# B&R Automation Studio project Nitto (part 8)

#### gunwfeedi.ax
```
InitParameter (Version=2.37.0, NcSwId=ACP10)
  ACP10AXIS_typ:
    dig_in:
      level:
        reference = ncACTIV_HI
        pos_hw_end = ncACTIV_HI
        neg_hw_end = ncACTIV_HI
        trigger1 = ncACTIV_HI
        trigger2 = ncACTIV_HI
    encoder_if:
      parameter:
        count_dir = ncSTANDARD
        scaling:
          load:
            units = 118000
            rev_motor = 83
    limit:
      parameter:
        v_pos = 75000.0
        v_neg = 75000.0
        a1_pos = 550000.0
        a2_pos = 550000.0
        a1_neg = 550000.0
        a2_neg = 550000.0
        t_jolt = 0.0
        t_in_pos = 0.0
        pos_sw_end = 2000000000
        neg_sw_end = -2000000000
        ds_warning = 1500.0
        ds_stop = 3000.0
        a_stop = 1.0e+30
        dv_stop = 0.0
        dv_stop_mode = ncOFF
    controller:
      mode = ncPOSITION
      position:
        kv = 50.0
        tn = 0.0
        t_predict = 0.002
        t_total = 0.002
        p_max = 1.0e+30
        i_max = 0.0
      speed:
        kv = 2.0
        tn = 0.0
        t_filter = 0.0
        isq_filter1:
          type = ncOFF
          a0 = 0.0
          a1 = 0.0
          b0 = 0.0
          b1 = 0.0
          b2 = 0.0
          c0_par_id = 0
          c1_par_id = 0
        isq_filter2:
          type = ncOFF
          a0 = 0.0
          a1 = 0.0
          b0 = 0.0
          b1 = 0.0
          b2 = 0.0
          c0_par_id = 0
          c1_par_id = 0
        isq_filter3:
          type = ncOFF
          a0 = 0.0
          a1 = 0.0
          b0 = 0.0
          b1 = 0.0
          b2 = 0.0
          c0_par_id = 0
          c1_par_id = 0
      uf:
        type = ncLINEAR
        auto_config = ncMOTOR_PAR
        u0 = 0.0
        un = 0.0
        fn = 50.0
        k_f_slip = 0.0
      ff:
        torque_load = 0.0
        torque_pos = 0.0
        torque_neg = 0.0
        kv_torque = 0.0
        inertia = 0.0
        t_filter_a = 0.0
    move:
      stop:
        parameter[0]:
          decel_ramp = ncA_LIMIT
          controller = ncON
        parameter[1]:
          decel_ramp = ncA_LIMIT
          controller = ncON
        parameter[2]:
          decel_ramp = ncA_LIMIT
          controller = ncON
        parameter[3]:
          decel_ramp = ncA_LIMIT
          controller = ncON
        quickstop:
          decel_ramp = ncA_LIMIT
        drive_error:
          decel_ramp = ncA_LIMIT
      homing:
        parameter:
          s = 0
          v_switch = 5000.0
          v_trigger = 500.0
          a = 50000.0
          mode = ncDIRECT
          edge_sw = ncPOSITIVE
          start_dir = ncPOSITIVE
          trigg_dir = ncPOSITIVE
          ref_pulse = ncOFF
          fix_dir = ncOFF
          tr_s_block = 0.0
          torque_lim = 0.0
          ds_block = 0.0
          ds_stop = 0.0
      basis:
        parameter:
          v_pos = 5000.0
          v_neg = 5000.0
          a1_pos = 100000.0
          a2_pos = 100000.0
          a1_neg = 100000.0
          a2_neg = 100000.0
    message:
      text:
        parameter:
          format = ncBREAK
          columns = 80
          data_modul = acp10etxen
```

### Data object Logical/AxisObj/ggrid1i (Ax)

#### ggrid1i.ax
```
InitParameter (Version=2.37.0, NcSwId=ACP10)
  ACP10AXIS_typ:
    dig_in:
      level:
        reference = ncACTIV_HI
        pos_hw_end = ncACTIV_HI
        neg_hw_end = ncACTIV_HI
        trigger1 = ncACTIV_HI
        trigger2 = ncACTIV_HI
    encoder_if:
      parameter:
        count_dir = ncSTANDARD
        scaling:
          load:
            units = 792000
            rev_motor = 2880
    limit:
      parameter:
        v_pos = 13750.0
        v_neg = 13750.0
        a1_pos = 46000.0
        a2_pos = 46000.0
        a1_neg = 46000.0
        a2_neg = 46000.0
        t_jolt = 0.0
        t_in_pos = 0.0
        pos_sw_end = 2000000000
        neg_sw_end = -2000000000
        ds_warning = 500.0
        ds_stop = 1000.0
        a_stop = 1.0e+30
        dv_stop = 0.0
        dv_stop_mode = ncOFF
    controller:
      mode = ncPOSITION
      position:
        kv = 180.0
        tn = 0.0
        t_predict = 0.0004
        t_total = 0.0004
        p_max = 1.0e+30
        i_max = 0.0
      speed:
        kv = 3.35
        tn = 0.0
        t_filter = 0.0
        isq_filter1:
          type = ncOFF
          a0 = 0.0
          a1 = 0.0
          b0 = 0.0
          b1 = 0.0
          b2 = 0.0
          c0_par_id = 0
          c1_par_id = 0
        isq_filter2:
          type = ncOFF
          a0 = 0.0
          a1 = 0.0
          b0 = 0.0
          b1 = 0.0
          b2 = 0.0
          c0_par_id = 0
          c1_par_id = 0
        isq_filter3:
          type = ncOFF
          a0 = 0.0
          a1 = 0.0
          b0 = 0.0
          b1 = 0.0
          b2 = 0.0
          c0_par_id = 0
          c1_par_id = 0
      uf:
        type = ncLINEAR
        auto_config = ncMOTOR_PAR
        u0 = 0.0
        un = 0.0
        fn = 50.0
        k_f_slip = 0.0
      ff:
        torque_load = 0.0
        torque_pos = 0.0
        torque_neg = 0.0
        kv_torque = 0.0
        inertia = 0.0
        t_filter_a = 0.0
    move:
      stop:
        parameter[0]:
          decel_ramp = ncA_LIMIT
          controller = ncON
        parameter[1]:
          decel_ramp = ncA_LIMIT
          controller = ncON
        parameter[2]:
          decel_ramp = ncA_LIMIT
          controller = ncON
        parameter[3]:
          decel_ramp = ncA_LIMIT
          controller = ncON
        quickstop:
          decel_ramp = ncA_LIMIT
        drive_error:
          decel_ramp = ncA_LIMIT
      homing:
        parameter:
          s = 0
          v_switch = 5000.0
          v_trigger = 500.0
          a = 50000.0
          mode = ncDIRECT
          edge_sw = ncPOSITIVE
          start_dir = ncPOSITIVE
          trigg_dir = ncPOSITIVE
          ref_pulse = ncOFF
          fix_dir = ncOFF
          tr_s_block = 0.0
          torque_lim = 0.0
          ds_block = 0.0
          ds_stop = 0.0
      basis:
        parameter:
          v_pos = 1000.0
          v_neg = 1000.0
          a1_pos = 1500.0
          a2_pos = 1500.0
          a1_neg = 1500.0
          a2_neg = 1500.0
    message:
      text:
        parameter:
          format = ncBREAK
          columns = 80
          data_modul = acp10etxen
```

### Data object Logical/AxisObj/ggrid2i (Ax)

#### ggrid2i.ax
```
InitParameter (Version=2.37.0, NcSwId=ACP10)
  ACP10AXIS_typ:
    dig_in:
      level:
        reference = ncACTIV_HI
        pos_hw_end = ncACTIV_HI
        neg_hw_end = ncACTIV_HI
        trigger1 = ncACTIV_HI
        trigger2 = ncACTIV_HI
    encoder_if:
      parameter:
        count_dir = ncINVERSE
        scaling:
          load:
            units = 1000
            rev_motor = 5
    limit:
      parameter:
        v_pos = 13750.0
        v_neg = 13750.0
        a1_pos = 46000.0
        a2_pos = 46000.0
        a1_neg = 46000.0
        a2_neg = 46000.0
        t_jolt = 0.0
        t_in_pos = 0.0
        pos_sw_end = 2000000000
        neg_sw_end = -2000000000
        ds_warning = 500.0
        ds_stop = 1000.0
        a_stop = 1.0e+30
        dv_stop = 0.0
        dv_stop_mode = ncOFF
    controller:
      mode = ncPOSITION
      position:
        kv = 140.0
        tn = 0.0
        t_predict = 0.0004
        t_total = 0.0004
        p_max = 1.0e+30
        i_max = 0.0
      speed:
        kv = 1.9
        tn = 0.0
        t_filter = 0.0
        isq_filter1:
          type = ncOFF
          a0 = 0.0
          a1 = 0.0
          b0 = 0.0
          b1 = 0.0
          b2 = 0.0
          c0_par_id = 0
          c1_par_id = 0
        isq_filter2:
          type = ncOFF
          a0 = 0.0
          a1 = 0.0
          b0 = 0.0
          b1 = 0.0
          b2 = 0.0
          c0_par_id = 0
          c1_par_id = 0
        isq_filter3:
          type = ncOFF
          a0 = 0.0
          a1 = 0.0
          b0 = 0.0
          b1 = 0.0
          b2 = 0.0
          c0_par_id = 0
          c1_par_id = 0
      uf:
        type = ncLINEAR
        auto_config = ncMOTOR_PAR
        u0 = 0.0
        un = 0.0
        fn = 50.0
        k_f_slip = 0.0
      ff:
        torque_load = 0.0
        torque_pos = 0.0
        torque_neg = 0.0
        kv_torque = 0.0
        inertia = 0.0
        t_filter_a = 0.0
    move:
      stop:
        parameter[0]:
          decel_ramp = ncA_LIMIT
          controller = ncON
        parameter[1]:
          decel_ramp = ncA_LIMIT
          controller = ncON
        parameter[2]:
          decel_ramp = ncA_LIMIT
          controller = ncON
        parameter[3]:
          decel_ramp = ncA_LIMIT
          controller = ncON
        quickstop:
          decel_ramp = ncA_LIMIT
        drive_error:
          decel_ramp = ncA_LIMIT
      homing:
        parameter:
          s = 0
          v_switch = 5000.0
          v_trigger = 500.0
          a = 50000.0
          mode = ncDIRECT
          edge_sw = ncPOSITIVE
          start_dir = ncPOSITIVE
          trigg_dir = ncPOSITIVE
          ref_pulse = ncOFF
          fix_dir = ncOFF
          tr_s_block = 0.0
          torque_lim = 0.0
          ds_block = 0.0
          ds_stop = 0.0
      basis:
        parameter:
          v_pos = 1000.0
          v_neg = 1000.0
          a1_pos = 1500.0
          a2_pos = 1500.0
          a1_neg = 1500.0
          a2_neg = 1500.0
    message:
      text:
        parameter:
          format = ncBREAK
          columns = 80
          data_modul = acp10etxen
```

### Data object Logical/AxisObj/gcut1i (Ax)

#### gcut1i.ax
```
InitParameter (Version=2.37.0, NcSwId=ACP10)
  ACP10AXIS_typ:
    dig_in:
      level:
        reference = ncACTIV_HI + ncFORCE
        pos_hw_end = ncACTIV_HI
        neg_hw_end = ncACTIV_HI
        trigger1 = ncACTIV_HI
        trigger2 = ncACTIV_HI
    encoder_if:
      parameter:
        count_dir = ncINVERSE
        scaling:
          load:
            units = 121920000
            rev_motor = 1200
    limit:
      parameter:
        v_pos = 833333.0
        v_neg = 833333.0
        a1_pos = 160000.0
        a2_pos = 160000.0
        a1_neg = 160000.0
        a2_neg = 160000.0
        t_jolt = 0.0
        t_in_pos = 0.0
        pos_sw_end = 8388607
        neg_sw_end = -8388608
        ds_warning = 25000.0
        ds_stop = 50000.0
        a_stop = 2.0e+10
        dv_stop = 100000.0
        dv_stop_mode = ncDV_STOP_INIT
    controller:
      mode = ncPOSITION
      position:
        kv = 400.0
        tn = 0.0
        t_predict = 0.0004
        t_total = 0.0004
        p_max = 1.0e+30
        i_max = 0.0
      speed:
        kv = 89.4
        tn = 0.0
        t_filter = 0.0
        isq_filter1:
          type = ncOFF
          a0 = 0.0
          a1 = 0.0
          b0 = 0.0
          b1 = 0.0
          b2 = 0.0
          c0_par_id = 0
          c1_par_id = 0
        isq_filter2:
          type = ncOFF
          a0 = 0.0
          a1 = 0.0
          b0 = 0.0
          b1 = 0.0
          b2 = 0.0
          c0_par_id = 0
          c1_par_id = 0
        isq_filter3:
          type = ncOFF
          a0 = 0.0
          a1 = 0.0
          b0 = 0.0
          b1 = 0.0
          b2 = 0.0
          c0_par_id = 0
          c1_par_id = 0
      uf:
        type = ncLINEAR
        auto_config = ncMOTOR_PAR
        u0 = 0.0
        un = 0.0
        fn = 50.0
        k_f_slip = 0.0
      ff:
        torque_load = 0.0
        torque_pos = 0.0
        torque_neg = 0.0
        kv_torque = 0.0
        inertia = 0.0
        t_filter_a = 0.0
    move:
      stop:
        parameter[0]:
          decel_ramp = ncA_LIMIT
          controller = ncON
        parameter[1]:
          decel_ramp = ncA_LIMIT
          controller = ncON
        parameter[2]:
          decel_ramp = ncA_LIMIT
          controller = ncON
        parameter[3]:
          decel_ramp = ncA_LIMIT
          controller = ncON
        quickstop:
          decel_ramp = ncA_LIMIT
        drive_error:
          decel_ramp = ncA_LIMIT
      homing:
        parameter:
          s = 230187
          v_switch = 20000.0
          v_trigger = 12700.0
          a = 60000.0
          mode = ncSWITCH_GATE
          edge_sw = ncPOSITIVE
          start_dir = ncPOSITIVE
          trigg_dir = ncPOSITIVE
          ref_pulse = ncOFF
          fix_dir = ncOFF
          tr_s_block = 0.0
          torque_lim = 0.0
          ds_block = 0.0
          ds_stop = 0.0
      basis:
        parameter:
          v_pos = 20000.0
          v_neg = 20000.0
          a1_pos = 60000.0
          a2_pos = 60000.0
          a1_neg = 60000.0
          a2_neg = 60000.0
    message:
      text:
        parameter:
          format = ncBREAK
          columns = 80
          data_modul = acp10etxde
```

### Data object Logical/AxisObj/gcut2i (Ax)

#### gcut2i.ax
```
InitParameter (Version=2.37.0, NcSwId=ACP10)
  ACP10AXIS_typ:
    dig_in:
      level:
        reference = ncACTIV_HI + ncFORCE
        pos_hw_end = ncACTIV_HI
        neg_hw_end = ncACTIV_HI
        trigger1 = ncACTIV_HI
        trigger2 = ncACTIV_HI
    encoder_if:
      parameter:
        count_dir = ncINVERSE
        scaling:
          load:
            units = 121920000
            rev_motor = 1200
    limit:
      parameter:
        v_pos = 833333.0
        v_neg = 833333.0
        a1_pos = 160000.0
        a2_pos = 160000.0
        a1_neg = 160000.0
        a2_neg = 160000.0
        t_jolt = 0.0
        t_in_pos = 0.0
        pos_sw_end = 8388607
        neg_sw_end = -8388608
        ds_warning = 25000.0
        ds_stop = 50000.0
        a_stop = 2.0e+10
        dv_stop = 100000.0
        dv_stop_mode = ncDV_STOP_INIT
    controller:
      mode = ncPOSITION
      position:
        kv = 400.0
        tn = 0.0
        t_predict = 0.0004
        t_total = 0.0004
        p_max = 1.0e+30
        i_max = 0.0
      speed:
        kv = 87.35
        tn = 0.0
        t_filter = 0.0
        isq_filter1:
          type = ncOFF
          a0 = 0.0
          a1 = 0.0
          b0 = 0.0
          b1 = 0.0
          b2 = 0.0
          c0_par_id = 0
          c1_par_id = 0
        isq_filter2:
          type = ncOFF
          a0 = 0.0
          a1 = 0.0
          b0 = 0.0
          b1 = 0.0
          b2 = 0.0
          c0_par_id = 0
          c1_par_id = 0
        isq_filter3:
          type = ncOFF
          a0 = 0.0
          a1 = 0.0
          b0 = 0.0
          b1 = 0.0
          b2 = 0.0
          c0_par_id = 0
          c1_par_id = 0
      uf:
        type = ncLINEAR
        auto_config = ncMOTOR_PAR
        u0 = 0.0
        un = 0.0
        fn = 50.0
        k_f_slip = 0.0
      ff:
        torque_load = 0.0
        torque_pos = 0.0
        torque_neg = 0.0
        kv_torque = 0.0
        inertia = 0.0
        t_filter_a = 0.0
    move:
      stop:
        parameter[0]:
          decel_ramp = ncA_LIMIT
          controller = ncON
        parameter[1]:
          decel_ramp = ncA_LIMIT
          controller = ncON
        parameter[2]:
          decel_ramp = ncA_LIMIT
          controller = ncON
        parameter[3]:
          decel_ramp = ncA_LIMIT
          controller = ncON
        quickstop:
          decel_ramp = ncA_LIMIT
        drive_error:
          decel_ramp = ncA_LIMIT
      homing:
        parameter:
          s = 0
          v_switch = 20000.0
          v_trigger = 12700.0
          a = 60000.0
          mode = ncSWITCH_GATE
          edge_sw = ncPOSITIVE
          start_dir = ncPOSITIVE
          trigg_dir = ncPOSITIVE
          ref_pulse = ncOFF
          fix_dir = ncOFF
          tr_s_block = 0.0
          torque_lim = 0.0
          ds_block = 0.0
          ds_stop = 0.0
      basis:
        parameter:
          v_pos = 20000.0
          v_neg = 20000.0
          a1_pos = 60000.0
          a2_pos = 60000.0
          a1_neg = 60000.0
          a2_neg = 60000.0
    message:
      text:
        parameter:
          format = ncBREAK
          columns = 80
          data_modul = acp10etxde
```

### Data object Logical/AxisObj/gmasteri (Vax)

- gmasteri.vax (not shown)

### Data object Logical/AxisObj/gpbs1i (Ax)

#### gpbs1i.ax
```
InitParameter (Version=2.37.0, NcSwId=ACP10)
  ACP10AXIS_typ:
    dig_in:
      level:
        reference = ncACTIV_HI
        pos_hw_end = ncACTIV_HI
        neg_hw_end = ncACTIV_HI
        trigger1 = ncACTIV_HI
        trigger2 = ncACTIV_HI
    encoder_if:
      parameter:
        count_dir = ncINVERSE
        scaling:
          load:
            units = 112588397
            rev_motor = 2000
    limit:
      parameter:
        v_pos = 833333.0
        v_neg = 833333.0
        a1_pos = 1676390.0
        a2_pos = 1676390.0
        a1_neg = 1676390.0
        a2_neg = 1676390.0
        t_jolt = 0.0
        t_in_pos = 0.0
        pos_sw_end = 2000000000
        neg_sw_end = -2000000000
        ds_warning = 15000.0
        ds_stop = 14000.0
        a_stop = 2.0e+08
        dv_stop = 0.0
        dv_stop_mode = ncOFF
    controller:
      mode = ncPOSITION
      position:
        kv = 240.0
        tn = 0.0
        t_predict = 0.0004
        t_total = 0.0004
        p_max = 1.0e+30
        i_max = 0.0
      speed:
        kv = 1.4
        tn = 0.0
        t_filter = 0.0008
        isq_filter1:
          type = ncOFF
          a0 = 0.0
          a1 = 0.0
          b0 = 0.0
          b1 = 0.0
          b2 = 0.0
          c0_par_id = 0
          c1_par_id = 0
        isq_filter2:
          type = ncOFF
          a0 = 0.0
          a1 = 0.0
          b0 = 0.0
          b1 = 0.0
          b2 = 0.0
          c0_par_id = 0
          c1_par_id = 0
        isq_filter3:
          type = ncOFF
          a0 = 0.0
          a1 = 0.0
          b0 = 0.0
          b1 = 0.0
          b2 = 0.0
          c0_par_id = 0
          c1_par_id = 0
      uf:
        type = ncLINEAR
        auto_config = ncMOTOR_PAR
        u0 = 0.0
        un = 0.0
        fn = 50.0
        k_f_slip = 0.0
      ff:
        torque_load = 0.0
        torque_pos = 0.539183
        torque_neg = 0.476101
        kv_torque = 0.027371
        inertia = 0.00657748
        t_filter_a = 0.0
    move:
      stop:
        parameter[0]:
          decel_ramp = ncA_LIMIT
          controller = ncON
        parameter[1]:
          decel_ramp = ncA_LIMIT
          controller = ncON
        parameter[2]:
          decel_ramp = ncA_LIMIT
          controller = ncON
        parameter[3]:
          decel_ramp = ncA_LIMIT
          controller = ncON
        quickstop:
          decel_ramp = ncA_LIMIT
        drive_error:
          decel_ramp = ncA_LIMIT
      homing:
        parameter:
          s = 0
          v_switch = 5000.0
          v_trigger = 500.0
          a = 50000.0
          mode = ncDIRECT
          edge_sw = ncPOSITIVE
          start_dir = ncPOSITIVE
          trigg_dir = ncPOSITIVE
          ref_pulse = ncOFF
          fix_dir = ncOFF
          tr_s_block = 0.0
          torque_lim = 0.0
          ds_block = 0.0
          ds_stop = 0.0
      basis:
        parameter:
          v_pos = 60000.0
          v_neg = 60000.0
          a1_pos = 100000.0
          a2_pos = 100000.0
          a1_neg = 100000.0
          a2_neg = 100000.0
    message:
      text:
        parameter:
          format = ncBREAK
          columns = 80
          data_modul = acp10etxde
```

### Data object Logical/AxisObj/gpbs2i (Ax)

#### gpbs2i.ax
```
InitParameter (Version=2.37.0, NcSwId=ACP10)
  ACP10AXIS_typ:
    dig_in:
      level:
        reference = ncACTIV_HI
        pos_hw_end = ncACTIV_HI
        neg_hw_end = ncACTIV_HI
        trigger1 = ncACTIV_HI
        trigger2 = ncACTIV_HI
    encoder_if:
      parameter:
        count_dir = ncINVERSE
        scaling:
          load:
            units = 5717683
            rev_motor = 370
    limit:
      parameter:
        v_pos = 833333.0
        v_neg = 833333.0
        a1_pos = 1651780.0
        a2_pos = 1651780.0
        a1_neg = 1651780.0
        a2_neg = 1651780.0
        t_jolt = 0.0
        t_in_pos = 0.0
        pos_sw_end = 2000000000
        neg_sw_end = -2000000000
        ds_warning = 15000.0
        ds_stop = 19000.0
        a_stop = 2.0e+08
        dv_stop = 0.0
        dv_stop_mode = ncOFF
    controller:
      mode = ncPOSITION
      position:
        kv = 340.0
        tn = 0.0
        t_predict = 0.0004
        t_total = 0.0004
        p_max = 1.0e+30
        i_max = 0.0
      speed:
        kv = 1.1
        tn = 0.0
        t_filter = 0.0008
        isq_filter1:
          type = ncOFF
          a0 = 0.0
          a1 = 0.0
          b0 = 0.0
          b1 = 0.0
          b2 = 0.0
          c0_par_id = 0
          c1_par_id = 0
        isq_filter2:
          type = ncOFF
          a0 = 0.0
          a1 = 0.0
          b0 = 0.0
          b1 = 0.0
          b2 = 0.0
          c0_par_id = 0
          c1_par_id = 0
        isq_filter3:
          type = ncOFF
          a0 = 0.0
          a1 = 0.0
          b0 = 0.0
          b1 = 0.0
          b2 = 0.0
          c0_par_id = 0
          c1_par_id = 0
      uf:
        type = ncLINEAR
        auto_config = ncMOTOR_PAR
        u0 = 0.0
        un = 0.0
        fn = 50.0
        k_f_slip = 0.0
      ff:
        torque_load = 0.0
        torque_pos = 0.539183
        torque_neg = 0.476101
        kv_torque = 0.027371
        inertia = 0.00657748
        t_filter_a = 0.0
    move:
      stop:
        parameter[0]:
          decel_ramp = ncA_LIMIT
          controller = ncON
        parameter[1]:
          decel_ramp = ncA_LIMIT
          controller = ncON
        parameter[2]:
          decel_ramp = ncA_LIMIT
          controller = ncON
        parameter[3]:
          decel_ramp = ncA_LIMIT
          controller = ncON
        quickstop:
          decel_ramp = ncA_LIMIT
        drive_error:
          decel_ramp = ncA_LIMIT
      homing:
        parameter:
          s = 0
          v_switch = 5000.0
          v_trigger = 500.0
          a = 50000.0
          mode = ncDIRECT
          edge_sw = ncPOSITIVE
          start_dir = ncPOSITIVE
          trigg_dir = ncPOSITIVE
          ref_pulse = ncOFF
          fix_dir = ncOFF
          tr_s_block = 0.0
          torque_lim = 0.0
          ds_block = 0.0
          ds_stop = 0.0
      basis:
        parameter:
          v_pos = 200000.0
          v_neg = 200000.0
          a1_pos = 10000.0
          a2_pos = 10000.0
          a1_neg = 10000.0
          a2_neg = 10000.0
    message:
      text:
        parameter:
          format = ncBREAK
          columns = 80
          data_modul = acp10etxde
```

### Data object Logical/AxisObj/gunwopi (Ax)

#### gunwopi.ax
```
InitParameter (Version=2.37.0, NcSwId=ACP10)
  ACP10AXIS_typ:
    dig_in:
      level:
        reference = ncACTIV_HI
        pos_hw_end = ncACTIV_HI
        neg_hw_end = ncACTIV_HI
        trigger1 = ncACTIV_HI
        trigger2 = ncACTIV_HI
    encoder_if:
      parameter:
        count_dir = ncSTANDARD
        scaling:
          load:
            units = 900000
            rev_motor = 7200
    limit:
      parameter:
        v_pos = 12500.0
        v_neg = 12500.0
        a1_pos = 100000.0
        a2_pos = 100000.0
        a1_neg = 100000.0
        a2_neg = 100000.0
        t_jolt = 0.0
        t_in_pos = 0.0
        pos_sw_end = 2000000000
        neg_sw_end = -2000000000
        ds_warning = 500.0
        ds_stop = 1000.0
        a_stop = 1.0e+30
        dv_stop = 0.0
        dv_stop_mode = ncOFF
    controller:
      mode = ncPOSITION
      position:
        kv = 240.0
        tn = 0.0
        t_predict = 0.0004
        t_total = 0.0004
        p_max = 1.0e+30
        i_max = 0.0
      speed:
        kv = 4.2
        tn = 0.0
        t_filter = 0.0
        isq_filter1:
          type = ncOFF
          a0 = 0.0
          a1 = 0.0
          b0 = 0.0
          b1 = 0.0
          b2 = 0.0
          c0_par_id = 0
          c1_par_id = 0
        isq_filter2:
          type = ncOFF
          a0 = 0.0
          a1 = 0.0
          b0 = 0.0
          b1 = 0.0
          b2 = 0.0
          c0_par_id = 0
          c1_par_id = 0
        isq_filter3:
          type = ncOFF
          a0 = 0.0
          a1 = 0.0
          b0 = 0.0
          b1 = 0.0
          b2 = 0.0
          c0_par_id = 0
          c1_par_id = 0
      uf:
        type = ncLINEAR
        auto_config = ncMOTOR_PAR
        u0 = 0.0
        un = 0.0
        fn = 50.0
        k_f_slip = 0.0
      ff:
        torque_load = 0.0
        torque_pos = 0.0
        torque_neg = 0.0
        kv_torque = 0.0
        inertia = 0.0
        t_filter_a = 0.0
    move:
      stop:
        parameter[0]:
          decel_ramp = ncA_LIMIT
          controller = ncON
        parameter[1]:
          decel_ramp = ncA_LIMIT
          controller = ncON
        parameter[2]:
          decel_ramp = ncA_LIMIT
          controller = ncON
        parameter[3]:
          decel_ramp = ncA_LIMIT
          controller = ncON
        quickstop:
          decel_ramp = ncA_LIMIT
        drive_error:
          decel_ramp = ncA_LIMIT
      homing:
        parameter:
          s = 0
          v_switch = 5000.0
          v_trigger = 500.0
          a = 50000.0
          mode = ncDIRECT
          edge_sw = ncPOSITIVE
          start_dir = ncPOSITIVE
          trigg_dir = ncPOSITIVE
          ref_pulse = ncOFF
          fix_dir = ncOFF
          tr_s_block = 0.0
          torque_lim = 0.0
          ds_block = 0.0
          ds_stop = 0.0
      basis:
        parameter:
          v_pos = 1000.0
          v_neg = 1000.0
          a1_pos = 5000.0
          a2_pos = 5000.0
          a1_neg = 5000.0
          a2_neg = 5000.0
    message:
      text:
        parameter:
          format = ncBREAK
          columns = 80
          data_modul = acp10etxen
```

### Data object Logical/AxisObj/gunwdrvi (Ax)

#### gunwdrvi.ax
```
InitParameter (Version=2.37.0, NcSwId=ACP10)
  ACP10AXIS_typ:
    dig_in:
      level:
        reference = ncACTIV_HI
        pos_hw_end = ncACTIV_HI
        neg_hw_end = ncACTIV_HI
        trigger1 = ncACTIV_HI
        trigger2 = ncACTIV_HI
    encoder_if:
      parameter:
        count_dir = ncINVERSE
        scaling:
          load:
            units = 900000
            rev_motor = 7200
    limit:
      parameter:
        v_pos = 12500.0
        v_neg = 12500.0
        a1_pos = 100000.0
        a2_pos = 100000.0
        a1_neg = 100000.0
        a2_neg = 100000.0
        t_jolt = 0.0
        t_in_pos = 0.0
        pos_sw_end = 2000000000
        neg_sw_end = -2000000000
        ds_warning = 500.0
        ds_stop = 1000.0
        a_stop = 1.0e+30
        dv_stop = 0.0
        dv_stop_mode = ncOFF
    controller:
      mode = ncPOSITION
      position:
        kv = 240.0
        tn = 0.0
        t_predict = 0.0004
        t_total = 0.0004
        p_max = 1.0e+30
        i_max = 0.0
      speed:
        kv = 4.0
        tn = 0.0
        t_filter = 0.0
        isq_filter1:
          type = ncOFF
          a0 = 0.0
          a1 = 0.0
          b0 = 0.0
          b1 = 0.0
          b2 = 0.0
          c0_par_id = 0
          c1_par_id = 0
        isq_filter2:
          type = ncOFF
          a0 = 0.0
          a1 = 0.0
          b0 = 0.0
          b1 = 0.0
          b2 = 0.0
          c0_par_id = 0
          c1_par_id = 0
        isq_filter3:
          type = ncOFF
          a0 = 0.0
          a1 = 0.0
          b0 = 0.0
          b1 = 0.0
          b2 = 0.0
          c0_par_id = 0
          c1_par_id = 0
      uf:
        type = ncLINEAR
        auto_config = ncMOTOR_PAR
        u0 = 0.0
        un = 0.0
        fn = 50.0
        k_f_slip = 0.0
      ff:
        torque_load = 0.0
        torque_pos = 0.0
        torque_neg = 0.0
        kv_torque = 0.0
        inertia = 0.0
        t_filter_a = 0.0
    move:
      stop:
        parameter[0]:
          decel_ramp = ncA_LIMIT
          controller = ncON
        parameter[1]:
          decel_ramp = ncA_LIMIT
          controller = ncON
        parameter[2]:
          decel_ramp = ncA_LIMIT
          controller = ncON
        parameter[3]:
          decel_ramp = ncA_LIMIT
          controller = ncON
        quickstop:
          decel_ramp = ncA_LIMIT
        drive_error:
          decel_ramp = ncA_LIMIT
      homing:
        parameter:
          s = 0
          v_switch = 5000.0
          v_trigger = 500.0
          a = 50000.0
          mode = ncDIRECT
          edge_sw = ncPOSITIVE
          start_dir = ncPOSITIVE
          trigg_dir = ncPOSITIVE
          ref_pulse = ncOFF
          fix_dir = ncOFF
          tr_s_block = 0.0
          torque_lim = 0.0
          ds_block = 0.0
          ds_stop = 0.0
      basis:
        parameter:
          v_pos = 1000.0
          v_neg = 1000.0
          a1_pos = 5000.0
          a2_pos = 5000.0
          a1_neg = 5000.0
          a2_neg = 5000.0
    message:
      text:
        parameter:
          format = ncBREAK
          columns = 80
          data_modul = acp10etxen
```

### Data object Logical/AxisObj/gcatchbi (Ax)

#### gcatchbi.ax
```
InitParameter (Version=2.37.0, NcSwId=ACP10)
  ACP10AXIS_typ:
    dig_in:
      level:
        reference = ncACTIV_HI
        pos_hw_end = ncACTIV_HI
        neg_hw_end = ncACTIV_HI
        trigger1 = ncACTIV_HI
        trigger2 = ncACTIV_HI
    encoder_if:
      parameter:
        count_dir = ncINVERSE
        scaling:
          load:
            units = 3777954
            rev_motor = 450
    limit:
      parameter:
        v_pos = 833333.0
        v_neg = 833333.0
        a1_pos = 1662110.0
        a2_pos = 1662110.0
        a1_neg = 1662110.0
        a2_neg = 1662110.0
        t_jolt = 0.0
        t_in_pos = 0.0
        pos_sw_end = 2000000000
        neg_sw_end = -2000000000
        ds_warning = 7000.0
        ds_stop = 8000.0
        a_stop = 2.0e+07
        dv_stop = 0.0
        dv_stop_mode = ncOFF
    controller:
      mode = ncPOSITION
      position:
        kv = 260.0
        tn = 0.0
        t_predict = 0.0004
        t_total = 0.0004
        p_max = 1.0e+30
        i_max = 0.0
      speed:
        kv = 0.15
        tn = 0.0
        t_filter = 0.0
        isq_filter1:
          type = ncOFF
          a0 = 0.0
          a1 = 0.0
          b0 = 0.0
          b1 = 0.0
          b2 = 0.0
          c0_par_id = 0
          c1_par_id = 0
        isq_filter2:
          type = ncOFF
          a0 = 0.0
          a1 = 0.0
          b0 = 0.0
          b1 = 0.0
          b2 = 0.0
          c0_par_id = 0
          c1_par_id = 0
        isq_filter3:
          type = ncOFF
          a0 = 0.0
          a1 = 0.0
          b0 = 0.0
          b1 = 0.0
          b2 = 0.0
          c0_par_id = 0
          c1_par_id = 0
      uf:
        type = ncLINEAR
        auto_config = ncMOTOR_PAR
        u0 = 0.0
        un = 0.0
        fn = 50.0
        k_f_slip = 0.0
      ff:
        torque_load = 0.0
        torque_pos = 0.0
        torque_neg = 0.0
        kv_torque = 0.0
        inertia = 0.0
        t_filter_a = 0.0
    move:
      stop:
        parameter[0]:
          decel_ramp = ncA_LIMIT
          controller = ncON
        parameter[1]:
          decel_ramp = ncA_LIMIT
          controller = ncON
        parameter[2]:
          decel_ramp = ncA_LIMIT
          controller = ncON
        parameter[3]:
          decel_ramp = ncA_LIMIT
          controller = ncON
        quickstop:
          decel_ramp = ncA_LIMIT
        drive_error:
          decel_ramp = ncA_LIMIT
      homing:
        parameter:
          s = 0
          v_switch = 5000.0
          v_trigger = 500.0
          a = 50000.0
          mode = ncDIRECT
          edge_sw = ncPOSITIVE
          start_dir = ncPOSITIVE
          trigg_dir = ncPOSITIVE
          ref_pulse = ncOFF
          fix_dir = ncOFF
          tr_s_block = 0.0
          torque_lim = 0.0
          ds_block = 0.0
          ds_stop = 0.0
      basis:
        parameter:
          v_pos = 100000.0
          v_neg = 500000.0
          a1_pos = 1000000.0
          a2_pos = 1000000.0
          a1_neg = 1000000.0
          a2_neg = 1000000.0
    message:
      text:
        parameter:
          format = ncBREAK
          columns = 80
          data_modul = acp10etxde
```

### Data object Logical/AxisObj/gconvbi (Ax)

#### gconvbi.ax
```
InitParameter (Version=2.37.0, NcSwId=ACP10)
  ACP10AXIS_typ:
    dig_in:
      level:
        reference = ncACTIV_HI
        pos_hw_end = ncACTIV_HI
        neg_hw_end = ncACTIV_HI
        trigger1 = ncACTIV_HI
        trigger2 = ncACTIV_HI
    encoder_if:
      parameter:
        count_dir = ncINVERSE
        scaling:
          load:
            units = 7796176
            rev_motor = 240
    limit:
      parameter:
        v_pos = 833333.0
        v_neg = 833333.0
        a1_pos = 1624200.0
        a2_pos = 1624200.0
        a1_neg = 1624200.0
        a2_neg = 1624200.0
        t_jolt = 0.0
        t_in_pos = 0.0
        pos_sw_end = 2000000000
        neg_sw_end = -2000000000
        ds_warning = 15000.0
        ds_stop = 16000.0
        a_stop = 2.0e+07
        dv_stop = 0.0
        dv_stop_mode = ncOFF
    controller:
      mode = ncPOSITION
      position:
        kv = 480.0
        tn = 0.0
        t_predict = 0.0004
        t_total = 0.0004
        p_max = 1.0e+30
        i_max = 0.0
      speed:
        kv = 0.6
        tn = 0.0
        t_filter = 0.0
        isq_filter1:
          type = ncOFF
          a0 = 0.0
          a1 = 0.0
          b0 = 0.0
          b1 = 0.0
          b2 = 0.0
          c0_par_id = 0
          c1_par_id = 0
        isq_filter2:
          type = ncOFF
          a0 = 0.0
          a1 = 0.0
          b0 = 0.0
          b1 = 0.0
          b2 = 0.0
          c0_par_id = 0
          c1_par_id = 0
        isq_filter3:
          type = ncOFF
          a0 = 0.0
          a1 = 0.0
          b0 = 0.0
          b1 = 0.0
          b2 = 0.0
          c0_par_id = 0
          c1_par_id = 0
      uf:
        type = ncLINEAR
        auto_config = ncMOTOR_PAR
        u0 = 0.0
        un = 0.0
        fn = 50.0
        k_f_slip = 0.0
      ff:
        torque_load = 0.0
        torque_pos = 0.0
        torque_neg = 0.0
        kv_torque = 0.0
        inertia = 0.0
        t_filter_a = 0.0
    move:
      stop:
        parameter[0]:
          decel_ramp = ncA_LIMIT
          controller = ncON
        parameter[1]:
          decel_ramp = ncA_LIMIT
          controller = ncON
        parameter[2]:
          decel_ramp = ncA_LIMIT
          controller = ncON
        parameter[3]:
          decel_ramp = ncA_LIMIT
          controller = ncON
        quickstop:
          decel_ramp = ncA_LIMIT
        drive_error:
          decel_ramp = ncA_LIMIT
      homing:
        parameter:
          s = 0
          v_switch = 5000.0
          v_trigger = 500.0
          a = 50000.0
          mode = ncDIRECT
          edge_sw = ncPOSITIVE
          start_dir = ncPOSITIVE
          trigg_dir = ncPOSITIVE
          ref_pulse = ncOFF
          fix_dir = ncOFF
          tr_s_block = 0.0
          torque_lim = 0.0
          ds_block = 0.0
          ds_stop = 0.0
      basis:
        parameter:
          v_pos = 500000.0
          v_neg = 100.0
          a1_pos = 1000000.0
          a2_pos = 1000000.0
          a1_neg = 1000000.0
          a2_neg = 1000000.0
    message:
      text:
        parameter:
          format = ncBREAK
          columns = 80
          data_modul = acp10etxde
```

### Data object Logical/AxisObj/glongcuti (Ax)

#### glongcuti.ax
```
InitParameter (Version=2.37.0, NcSwId=ACP10)
  ACP10AXIS_typ:
    dig_in:
      level:
        reference = ncACTIV_HI
        pos_hw_end = ncACTIV_HI
        neg_hw_end = ncACTIV_HI
        trigger1 = ncACTIV_HI
        trigger2 = ncACTIV_HI
    encoder_if:
      parameter:
        count_dir = ncINVERSE
        scaling:
          load:
            units = 13524556
            rev_motor = 410
    limit:
      parameter:
        v_pos = 833333.0
        v_neg = 833333.0
        a1_pos = 1649340.0
        a2_pos = 1649340.0
        a1_neg = 1649340.0
        a2_neg = 1649340.0
        t_jolt = 0.0
        t_in_pos = 0.0
        pos_sw_end = 2000000000
        neg_sw_end = -2000000000
        ds_warning = 15000.0
        ds_stop = 16500.0
        a_stop = 2.0e+07
        dv_stop = 100000.0
        dv_stop_mode = ncDV_STOP_INIT
    controller:
      mode = ncPOSITION
      position:
        kv = 540.0
        tn = 0.0
        t_predict = 0.0004
        t_total = 0.0004
        p_max = 1.0e+30
        i_max = 0.0
      speed:
        kv = 0.3
        tn = 0.0
        t_filter = 0.0
        isq_filter1:
          type = ncOFF
          a0 = 0.0
          a1 = 0.0
          b0 = 0.0
          b1 = 0.0
          b2 = 0.0
          c0_par_id = 0
          c1_par_id = 0
        isq_filter2:
          type = ncOFF
          a0 = 0.0
          a1 = 0.0
          b0 = 0.0
          b1 = 0.0
          b2 = 0.0
          c0_par_id = 0
          c1_par_id = 0
        isq_filter3:
          type = ncOFF
          a0 = 0.0
          a1 = 0.0
          b0 = 0.0
          b1 = 0.0
          b2 = 0.0
          c0_par_id = 0
          c1_par_id = 0
      uf:
        type = ncLINEAR
        auto_config = ncMOTOR_PAR
        u0 = 0.0
        un = 0.0
        fn = 50.0
        k_f_slip = 0.0
      ff:
        torque_load = 0.0
        torque_pos = 0.0
        torque_neg = 0.0
        kv_torque = 0.0
        inertia = 0.0
        t_filter_a = 0.0
    move:
      stop:
        parameter[0]:
          decel_ramp = ncA_LIMIT
          controller = ncON
        parameter[1]:
          decel_ramp = ncA_LIMIT
          controller = ncON
        parameter[2]:
          decel_ramp = ncA_LIMIT
          controller = ncON
        parameter[3]:
          decel_ramp = ncA_LIMIT
          controller = ncON
        quickstop:
          decel_ramp = ncA_LIMIT
        drive_error:
          decel_ramp = ncA_LIMIT
      homing:
        parameter:
          s = 0
          v_switch = 5000.0
          v_trigger = 500.0
          a = 50000.0
          mode = ncDIRECT
          edge_sw = ncPOSITIVE
          start_dir = ncPOSITIVE
          trigg_dir = ncPOSITIVE
          ref_pulse = ncOFF
          fix_dir = ncOFF
          tr_s_block = 0.0
          torque_lim = 0.0
          ds_block = 0.0
          ds_stop = 0.0
      basis:
        parameter:
          v_pos = 20000.0
          v_neg = 20000.0
          a1_pos = 250000.0
          a2_pos = 250000.0
          a1_neg = 250000.0
          a2_neg = 250000.0
    message:
      text:
        parameter:
          format = ncBREAK
          columns = 80
          data_modul = acp10etxen
```

### Data object Logical/AxisObj/ggridfeedi (Ax) - ACP10: Achse Datenobjekt.

#### ggridfeedi.ax
```
InitParameter (Version=2.37.0, NcSwId=ACP10)
  ACP10AXIS_typ:
    dig_in:
      level:
        reference = ncACTIV_HI
        pos_hw_end = ncACTIV_HI
        neg_hw_end = ncACTIV_HI
        trigger1 = ncACTIV_HI
        trigger2 = ncACTIV_HI
    encoder_if:
      parameter:
        count_dir = ncINVERSE
        scaling:
          load:
            units = 24480000
            rev_motor = 8174
    limit:
      parameter:
        v_pos = 833333.0
        v_neg = 833333.0
        a1_pos = 435584.0
        a2_pos = 435584.0
        a1_neg = 435584.0
        a2_neg = 435584.0
        t_jolt = 0.0
        t_in_pos = 0.0
        pos_sw_end = 2000000000
        neg_sw_end = -2000000000
        ds_warning = 80000.0
        ds_stop = 130000.0
        a_stop = 2.0e+10
        dv_stop = 10000.0
        dv_stop_mode = ncDV_STOP_INIT
    controller:
      mode = ncPOSITION
      position:
        kv = 50.0
        tn = 0.0
        t_predict = 0.0004
        t_total = 0.0004
        p_max = 10000.0
        i_max = 0.0
      speed:
        kv = 2.0
        tn = 0.0
        t_filter = 0.0
        isq_filter1:
          type = ncOFF
          a0 = 0.0
          a1 = 0.0
          b0 = 0.0
          b1 = 0.0
          b2 = 0.0
          c0_par_id = 0
          c1_par_id = 0
        isq_filter2:
          type = ncOFF
          a0 = 0.0
          a1 = 0.0
          b0 = 0.0
          b1 = 0.0
          b2 = 0.0
          c0_par_id = 0
          c1_par_id = 0
        isq_filter3:
          type = ncOFF
          a0 = 0.0
          a1 = 0.0
          b0 = 0.0
          b1 = 0.0
          b2 = 0.0
          c0_par_id = 0
          c1_par_id = 0
      uf:
        type = ncLINEAR
        auto_config = ncMOTOR_PAR
        u0 = 0.0
        un = 0.0
        fn = 50.0
        k_f_slip = 0.0
      ff:
        torque_load = 0.0
        torque_pos = 0.0
        torque_neg = 0.0
        kv_torque = 0.0
        inertia = 0.0
        t_filter_a = 0.0
    move:
      stop:
        parameter[0]:
          decel_ramp = ncA_LIMIT
          controller = ncON
        parameter[1]:
          decel_ramp = ncA_LIMIT
          controller = ncON
        parameter[2]:
          decel_ramp = ncA_LIMIT
          controller = ncON
        parameter[3]:
          decel_ramp = ncA_LIMIT
          controller = ncON
        quickstop:
          decel_ramp = ncA_LIMIT
        drive_error:
          decel_ramp = ncA_LIMIT
      homing:
        parameter:
          s = 0
          v_switch = 10000.0
          v_trigger = 1000.0
          a = 50000.0
          mode = ncABS_SWITCH
          edge_sw = ncPOSITIVE
          start_dir = ncPOSITIVE
          trigg_dir = ncNEGATIVE
          ref_pulse = ncOFF
          fix_dir = ncOFF
          tr_s_block = 0.0
          torque_lim = 0.0
          ds_block = 0.0
          ds_stop = 0.0
      basis:
        parameter:
          v_pos = 2000.0
          v_neg = 2000.0
          a1_pos = 10000.0
          a2_pos = 10000.0
          a1_neg = 10000.0
          a2_neg = 10000.0
    message:
      text:
        parameter:
          format = ncBREAK
          columns = 80
          data_modul = acp10etxde
```

### Data object Logical/AxisObj/gbufferi (Ax) - ACP10: Achse Datenobjekt.

#### gbufferi.ax
```
InitParameter (Version=2.37.0, NcSwId=ACP10)
  ACP10AXIS_typ:
    dig_in:
      level:
        reference = ncACTIV_HI
        pos_hw_end = ncACTIV_HI + ncFORCE
        neg_hw_end = ncACTIV_HI + ncFORCE
        trigger1 = ncACTIV_HI
        trigger2 = ncACTIV_HI
    encoder_if:
      parameter:
        count_dir = ncSTANDARD
        scaling:
          load:
            units = 1320000
            rev_motor = 15840
    limit:
      parameter:
        v_pos = 4166.0
        v_neg = 4166.0
        a1_pos = 41666.0
        a2_pos = 41666.0
        a1_neg = 41666.0
        a2_neg = 41666.0
        t_jolt = 0.0
        t_in_pos = 0.0
        pos_sw_end = 6550
        neg_sw_end = -10
        ds_warning = 10000.0
        ds_stop = 5000.0
        a_stop = 1.0e+30
        dv_stop = 0.0
        dv_stop_mode = ncOFF
    controller:
      mode = ncPOSITION + ncFF
      position:
        kv = 380.0
        tn = 0.0
        t_predict = 0.0004
        t_total = 0.0004
        p_max = 1.0e+30
        i_max = 0.0
      speed:
        kv = 10.25
        tn = 0.0
        t_filter = 0.0
        isq_filter1:
          type = ncOFF
          a0 = 0.0
          a1 = 0.0
          b0 = 0.0
          b1 = 0.0
          b2 = 0.0
          c0_par_id = 0
          c1_par_id = 0
        isq_filter2:
          type = ncOFF
          a0 = 0.0
          a1 = 0.0
          b0 = 0.0
          b1 = 0.0
          b2 = 0.0
          c0_par_id = 0
          c1_par_id = 0
        isq_filter3:
          type = ncOFF
          a0 = 0.0
          a1 = 0.0
          b0 = 0.0
          b1 = 0.0
          b2 = 0.0
          c0_par_id = 0
          c1_par_id = 0
      uf:
        type = ncLINEAR
        auto_config = ncMOTOR_PAR
        u0 = 0.0
        un = 0.0
        fn = 50.0
        k_f_slip = 0.0
      ff:
        torque_load = 1.23348
        torque_pos = 0.378458
        torque_neg = 0.355359
        kv_torque = 0.650491
        inertia = 0.0
        t_filter_a = 0.0
    move:
      stop:
        parameter[0]:
          decel_ramp = ncA_LIMIT
          controller = ncON
        parameter[1]:
          decel_ramp = ncA_LIMIT
          controller = ncON
        parameter[2]:
          decel_ramp = ncA_LIMIT
          controller = ncON
        parameter[3]:
          decel_ramp = ncA_LIMIT
          controller = ncON
        quickstop:
          decel_ramp = ncA_LIMIT
        drive_error:
          decel_ramp = ncA_LIMIT
      homing:
        parameter:
          s = 0
          v_switch = 100.0
          v_trigger = 40.0
          a = 1000.0
          mode = ncEND_SWITCH
          edge_sw = ncNEGATIVE
          start_dir = ncNEGATIVE
          trigg_dir = ncNEGATIVE
          ref_pulse = ncOFF
          fix_dir = ncOFF
          tr_s_block = 0.0
          torque_lim = 1.0
          ds_block = 0.0
          ds_stop = 0.0
      basis:
        parameter:
          v_pos = 200.0
          v_neg = 100.0
          a1_pos = 2000.0
          a2_pos = 2000.0
          a1_neg = 2000.0
          a2_neg = 2000.0
    message:
      text:
        parameter:
          format = ncBREAK
          columns = 80
          data_modul = acp10etxde
```

### Data object Logical/AxisObj/gPackBelti (Ax)

#### gPackBelti.ax
```
InitParameter (Version=2.37.0, NcSwId=ACP10)
  ACP10AXIS_typ:
    dig_in:
      level:
        reference = ncACTIV_HI
        pos_hw_end = ncACTIV_HI
        neg_hw_end = ncACTIV_HI
        trigger1 = ncACTIV_HI
        trigger2 = ncACTIV_HI
    encoder_if:
      parameter:
        count_dir = ncSTANDARD
        scaling:
          load:
            units = 118000
            rev_motor = 1
    limit:
      parameter:
        v_pos = 75000.0
        v_neg = 75000.0
        a1_pos = 550000.0
        a2_pos = 550000.0
        a1_neg = 550000.0
        a2_neg = 550000.0
        t_jolt = 0.0
        t_in_pos = 0.0
        pos_sw_end = 2000000000
        neg_sw_end = -2000000000
        ds_warning = 1000000.0
        ds_stop = 2000000.0
        a_stop = 1.0e+30
        dv_stop = 0.0
        dv_stop_mode = ncOFF
    controller:
      mode = ncPOSITION
      position:
        kv = 50.0
        tn = 0.0
        t_predict = 0.004
        t_total = 0.004
        p_max = 1.0e+30
        i_max = 0.0
      speed:
        kv = 2.0
        tn = 0.0
        t_filter = 0.0
        isq_filter1:
          type = ncOFF
          a0 = 0.0
          a1 = 0.0
          b0 = 0.0
          b1 = 0.0
          b2 = 0.0
          c0_par_id = 0
          c1_par_id = 0
        isq_filter2:
          type = ncOFF
          a0 = 0.0
          a1 = 0.0
          b0 = 0.0
          b1 = 0.0
          b2 = 0.0
          c0_par_id = 0
          c1_par_id = 0
        isq_filter3:
          type = ncOFF
          a0 = 0.0
          a1 = 0.0
          b0 = 0.0
          b1 = 0.0
          b2 = 0.0
          c0_par_id = 0
          c1_par_id = 0
      uf:
        type = ncLINEAR
        auto_config = ncMOTOR_PAR
        u0 = 0.0
        un = 0.0
        fn = 50.0
        k_f_slip = 0.0
      ff:
        torque_load = 0.0
        torque_pos = 0.0
        torque_neg = 0.0
        kv_torque = 0.0
        inertia = 0.0
        t_filter_a = 0.0
    move:
      stop:
        parameter[0]:
          decel_ramp = ncA_LIMIT
          controller = ncON
        parameter[1]:
          decel_ramp = ncA_LIMIT
          controller = ncON
        parameter[2]:
          decel_ramp = ncA_LIMIT
          controller = ncON
        parameter[3]:
          decel_ramp = ncA_LIMIT
          controller = ncON
        quickstop:
          decel_ramp = ncA_LIMIT
        drive_error:
          decel_ramp = ncA_LIMIT
      homing:
        parameter:
          s = 0
          v_switch = 5000.0
          v_trigger = 500.0
          a = 50000.0
          mode = ncDIRECT
          edge_sw = ncPOSITIVE
          start_dir = ncPOSITIVE
          trigg_dir = ncPOSITIVE
          ref_pulse = ncOFF
          fix_dir = ncOFF
          tr_s_block = 0.0
          torque_lim = 0.0
          ds_block = 0.0
          ds_stop = 0.0
      basis:
        parameter:
          v_pos = 1000.0
          v_neg = 1000.0
          a1_pos = 10000.0
          a2_pos = 10000.0
          a1_neg = 10000.0
          a2_neg = 10000.0
    message:
      text:
        parameter:
          format = ncBREAK
          columns = 80
          data_modul = acp10etxde
```

### Data object Logical/AxisObj/gconvbelta (Apt)

#### gconvbelta.apt
```
AcoposParameterTable:
  Root Parameters:
    390 = 560 (Name=UDC_NOMINAL, Unit=V)  // CTRL DC bus: Nominal voltage
    128 = 1 (Name=SGEN_SW_END_IGNORE)  // Limit values: Ignore SW end positions
    M1 (StructureEdit=FALSE)  // 8LSA36.R0060D000-0
      Allgemeine Parameter:
        30 = 16#0002 (Name=MOTOR_TYPE)  // Motor: Type
        31 = 16#0203 (Name=MOTOR_COMPATIBILITY)  // Motor: Software compatibility
        46 = 1 (Name=MOTOR_WIND_CONNECT)  // Motor: Winding connection
        47 = 2 (Name=MOTOR_POLEPAIRS)  // Motor: Number of pole-pairs
      Bremsparameter:
        42 = 0 (Name=MOTOR_BRAKE_CURR_RATED, Unit=A)  // Motor holding brake: Rated current
        43 = 0 (Name=MOTOR_BRAKE_TORQ_RATED, Unit=Nm)  // Motor holding brake: Rated torque
        44 = 0 (Name=MOTOR_BRAKE_ON_TIME, Unit=s)  // Motor holding brake: Engaging delay
        45 = 0 (Name=MOTOR_BRAKE_OFF_TIME, Unit=s)  // Motor holding brake: Release delay
      Thermosensor Parameter:
        64 = 632 (Name=MOTOR_TEMPSENS_PAR1)  // Temperature sensor: Parameter 1
        65 = 2225 (Name=MOTOR_TEMPSENS_PAR2)  // Temperature sensor: Parameter 2
        66 = -30 (Name=MOTOR_TEMPSENS_PAR3)  // Temperature sensor: Parameter 3
        67 = 5.7266 (Name=MOTOR_TEMPSENS_PAR4)  // Temperature sensor: Parameter 4
        68 = 36.0938 (Name=MOTOR_TEMPSENS_PAR5)  // Temperature sensor: Parameter 5
        69 = 62.9375 (Name=MOTOR_TEMPSENS_PAR6)  // Temperature sensor: Parameter 6
        70 = 87.25 (Name=MOTOR_TEMPSENS_PAR7)  // Temperature sensor: Parameter 7
        71 = 109.6016 (Name=MOTOR_TEMPSENS_PAR8)  // Temperature sensor: Parameter 8
        72 = 130.3984 (Name=MOTOR_TEMPSENS_PAR9)  // Temperature sensor: Parameter 9
        73 = 150 (Name=MOTOR_TEMPSENS_PAR10)  // Temperature sensor: Parameter 10
      Motorparameter:
        48 = 400 (Name=MOTOR_VOLTAGE_RATED, Unit=V)  // Motor: Rated voltage
        49 = 43.98 (Name=MOTOR_VOLTAGE_CONST, Unit=mV*min)  // Motor: Voltage constant
        50 = 6000 (Name=MOTOR_SPEED_RATED, Unit=1/min)  // Motor: Rated speed
        51 = 12000 (Name=MOTOR_SPEED_MAX, Unit=1/min)  // Motor: Maximum speed
        52 = 3 (Name=MOTOR_TORQ_STALL, Unit=Nm)  // Motor: Stall torque
        53 = 1.8 (Name=MOTOR_TORQ_RATED, Unit=Nm)  // Motor: Rated torque
        54 = 12 (Name=MOTOR_TORQ_MAX, Unit=Nm)  // Motor: Peak torque
        55 = 0.73 (Name=MOTOR_TORQ_CONST, Unit=Nm/A)  // Motor: Torque constant
        56 = 4.12 (Name=MOTOR_CURR_STALL, Unit=A)  // Motor: Stall current
        57 = 2.47 (Name=MOTOR_CURR_RATED, Unit=A)  // Motor: Rated current
        58 = 17.73 (Name=MOTOR_CURR_MAX, Unit=A)  // Motor: Peak current
        59 = 0.454 (Name=MOTOR_WIND_CROSS_SECT, Unit=mm²)  // Motor: Line cross section
        60 = 2.9 (Name=MOTOR_STATOR_RESISTANCE, Unit=Ohm)  // Motor: Stator resistance
        61 = 0.00945 (Name=MOTOR_STATOR_INDUCTANCE, Unit=Henry)  // Motor: Stator inductance
        62 = 0.00012 (Name=MOTOR_INERTIA, Unit=kgm²)  // Motor: Moment of inertia
        63 = 0 (Name=MOTOR_COMMUT_OFFSET, Unit=rad)  // Motor: Commutation offset
        849 = 2400 (Name=MOTOR_TAU_THERM, Unit=s)  // Motor: Thermal time constant
      Isolations Parameter:
        74 = 130 (Name=MOTOR_WIND_TEMP_MAX, Unit=°C)  // Motor: Limit temperature
```

### Data object Logical/AxisObj/gpbs2a (Apt)

#### gpbs2a.apt
```
AcoposParameterTable:
  Root Parameters:
    M1 (StructureEdit=FALSE)  // 8LSA43.R0045D000-0
      Allgemeine Parameter:
        30 = 16#0002 (Name=MOTOR_TYPE)  // Motor: Type
        31 = 16#0203 (Name=MOTOR_COMPATIBILITY)  // Motor: Software compatibility
        46 = 1 (Name=MOTOR_WIND_CONNECT)  // Motor: Winding connection
        47 = 5 (Name=MOTOR_POLEPAIRS)  // Motor: Number of pole-pairs
      Bremsparameter:
        42 = 0 (Name=MOTOR_BRAKE_CURR_RATED, Unit=A)  // Motor holding brake: Rated current
        43 = 0 (Name=MOTOR_BRAKE_TORQ_RATED, Unit=Nm)  // Motor holding brake: Rated torque
        44 = 0 (Name=MOTOR_BRAKE_ON_TIME, Unit=s)  // Motor holding brake: Engaging delay
        45 = 0 (Name=MOTOR_BRAKE_OFF_TIME, Unit=s)  // Motor holding brake: Release delay
      Thermosensor Parameter:
        64 = 632 (Name=MOTOR_TEMPSENS_PAR1)  // Temperature sensor: Parameter 1
        65 = 2225 (Name=MOTOR_TEMPSENS_PAR2)  // Temperature sensor: Parameter 2
        66 = -30 (Name=MOTOR_TEMPSENS_PAR3)  // Temperature sensor: Parameter 3
        67 = 5.7266 (Name=MOTOR_TEMPSENS_PAR4)  // Temperature sensor: Parameter 4
        68 = 36.0938 (Name=MOTOR_TEMPSENS_PAR5)  // Temperature sensor: Parameter 5
        69 = 62.9375 (Name=MOTOR_TEMPSENS_PAR6)  // Temperature sensor: Parameter 6
        70 = 87.25 (Name=MOTOR_TEMPSENS_PAR7)  // Temperature sensor: Parameter 7
        71 = 109.6016 (Name=MOTOR_TEMPSENS_PAR8)  // Temperature sensor: Parameter 8
        72 = 130.3984 (Name=MOTOR_TEMPSENS_PAR9)  // Temperature sensor: Parameter 9
        73 = 150 (Name=MOTOR_TEMPSENS_PAR10)  // Temperature sensor: Parameter 10
      Motorparameter:
        48 = 400 (Name=MOTOR_VOLTAGE_RATED, Unit=V)  // Motor: Rated voltage
        49 = 65.97 (Name=MOTOR_VOLTAGE_CONST, Unit=mV*min)  // Motor: Voltage constant
        50 = 4500 (Name=MOTOR_SPEED_RATED, Unit=1/min)  // Motor: Rated speed
        51 = 12000 (Name=MOTOR_SPEED_MAX, Unit=1/min)  // Motor: Maximum speed
        52 = 4 (Name=MOTOR_TORQ_STALL, Unit=Nm)  // Motor: Stall torque
        53 = 2.7 (Name=MOTOR_TORQ_RATED, Unit=Nm)  // Motor: Rated torque
        54 = 15.2 (Name=MOTOR_TORQ_MAX, Unit=Nm)  // Motor: Peak torque
        55 = 1.08 (Name=MOTOR_TORQ_CONST, Unit=Nm/A)  // Motor: Torque constant
        56 = 3.69 (Name=MOTOR_CURR_STALL, Unit=A)  // Motor: Stall current
        57 = 2.49 (Name=MOTOR_CURR_RATED, Unit=A)  // Motor: Rated current
        58 = 21.94 (Name=MOTOR_CURR_MAX, Unit=A)  // Motor: Peak current
        59 = 0.5027 (Name=MOTOR_WIND_CROSS_SECT, Unit=mm²)  // Motor: Line cross section
        60 = 2.64 (Name=MOTOR_STATOR_RESISTANCE, Unit=Ohm)  // Motor: Stator resistance
        61 = 0.0165 (Name=MOTOR_STATOR_INDUCTANCE, Unit=Henry)  // Motor: Stator inductance
        62 = 0.000187 (Name=MOTOR_INERTIA, Unit=kgm²)  // Motor: Moment of inertia
        63 = 0 (Name=MOTOR_COMMUT_OFFSET, Unit=rad)  // Motor: Commutation offset
        849 = 1500 (Name=MOTOR_TAU_THERM, Unit=s)  // Motor: Thermal time constant
      Isolations Parameter:
        74 = 130 (Name=MOTOR_WIND_TEMP_MAX, Unit=°C)  // Motor: Limit temperature
    390 = 560 (Name=UDC_NOMINAL, Unit=V)  // CTRL DC bus: Nominal voltage
    128 = 1 (Name=SGEN_SW_END_IGNORE)  // Limit values: Ignore SW end positions
```

### Data object Logical/AxisObj/gpbs1a (Apt)

#### gpbs1a.apt
```
AcoposParameterTable:
  Root Parameters:
    128 = 1 (Name=SGEN_SW_END_IGNORE)  // Limit values: Ignore SW end positions
    390 = 560 (Name=UDC_NOMINAL, Unit=V)  // CTRL DC bus: Nominal voltage
    M1 (StructureEdit=FALSE)  // 8LSA46.R0045D000-0
      Allgemeine Parameter:
        30 = 16#0002 (Name=MOTOR_TYPE)  // Motor: Type
        31 = 16#0203 (Name=MOTOR_COMPATIBILITY)  // Motor: Software compatibility
        46 = 1 (Name=MOTOR_WIND_CONNECT)  // Motor: Winding connection
        47 = 5 (Name=MOTOR_POLEPAIRS)  // Motor: Number of pole-pairs
      Bremsparameter:
        42 = 0 (Name=MOTOR_BRAKE_CURR_RATED, Unit=A)  // Motor holding brake: Rated current
        43 = 0 (Name=MOTOR_BRAKE_TORQ_RATED, Unit=Nm)  // Motor holding brake: Rated torque
        44 = 0 (Name=MOTOR_BRAKE_ON_TIME, Unit=s)  // Motor holding brake: Engaging delay
        45 = 0 (Name=MOTOR_BRAKE_OFF_TIME, Unit=s)  // Motor holding brake: Release delay
      Thermosensor Parameter:
        64 = 632 (Name=MOTOR_TEMPSENS_PAR1)  // Temperature sensor: Parameter 1
        65 = 2225 (Name=MOTOR_TEMPSENS_PAR2)  // Temperature sensor: Parameter 2
        66 = -30 (Name=MOTOR_TEMPSENS_PAR3)  // Temperature sensor: Parameter 3
        67 = 5.7266 (Name=MOTOR_TEMPSENS_PAR4)  // Temperature sensor: Parameter 4
        68 = 36.0938 (Name=MOTOR_TEMPSENS_PAR5)  // Temperature sensor: Parameter 5
        69 = 62.9375 (Name=MOTOR_TEMPSENS_PAR6)  // Temperature sensor: Parameter 6
        70 = 87.25 (Name=MOTOR_TEMPSENS_PAR7)  // Temperature sensor: Parameter 7
        71 = 109.6016 (Name=MOTOR_TEMPSENS_PAR8)  // Temperature sensor: Parameter 8
        72 = 130.3984 (Name=MOTOR_TEMPSENS_PAR9)  // Temperature sensor: Parameter 9
        73 = 150 (Name=MOTOR_TEMPSENS_PAR10)  // Temperature sensor: Parameter 10
      Motorparameter:
        48 = 400 (Name=MOTOR_VOLTAGE_RATED, Unit=V)  // Motor: Rated voltage
        49 = 65.97 (Name=MOTOR_VOLTAGE_CONST, Unit=mV*min)  // Motor: Voltage constant
        50 = 4500 (Name=MOTOR_SPEED_RATED, Unit=1/min)  // Motor: Rated speed
        51 = 12000 (Name=MOTOR_SPEED_MAX, Unit=1/min)  // Motor: Maximum speed
        52 = 10 (Name=MOTOR_TORQ_STALL, Unit=Nm)  // Motor: Stall torque
        53 = 6 (Name=MOTOR_TORQ_RATED, Unit=Nm)  // Motor: Rated torque
        54 = 38 (Name=MOTOR_TORQ_MAX, Unit=Nm)  // Motor: Peak torque
        55 = 1.08 (Name=MOTOR_TORQ_CONST, Unit=Nm/A)  // Motor: Torque constant
        56 = 9.24 (Name=MOTOR_CURR_STALL, Unit=A)  // Motor: Stall current
        57 = 5.54 (Name=MOTOR_CURR_RATED, Unit=A)  // Motor: Rated current
        58 = 54.85 (Name=MOTOR_CURR_MAX, Unit=A)  // Motor: Peak current
        59 = 1.272 (Name=MOTOR_WIND_CROSS_SECT, Unit=mm²)  // Motor: Line cross section
        60 = 0.8 (Name=MOTOR_STATOR_RESISTANCE, Unit=Ohm)  // Motor: Stator resistance
        61 = 0.00775 (Name=MOTOR_STATOR_INDUCTANCE, Unit=Henry)  // Motor: Stator inductance
        62 = 0.000439 (Name=MOTOR_INERTIA, Unit=kgm²)  // Motor: Moment of inertia
        63 = 0 (Name=MOTOR_COMMUT_OFFSET, Unit=rad)  // Motor: Commutation offset
        849 = 2400 (Name=MOTOR_TAU_THERM, Unit=s)  // Motor: Thermal time constant
      Isolations Parameter:
        74 = 130 (Name=MOTOR_WIND_TEMP_MAX, Unit=°C)  // Motor: Limit temperature
```

### Data object Logical/AxisObj/gunwa (Apt)

#### gunwopa.apt
```
AcoposParameterTable:
  Root Parameters:
    128 = 1 (Name=SGEN_SW_END_IGNORE)  // Limit values: Ignore SW end positions
    390 = 560 (Name=UDC_NOMINAL, Unit=V)  // CTRL DC bus: Nominal voltage
    M1 (StructureEdit=FALSE)  // 8LSN45.R0060D100-0
      Allgemeine Parameter:
        30 = 16#0002 (Name=MOTOR_TYPE)  // Motor: Type
        31 = 16#0203 (Name=MOTOR_COMPATIBILITY)  // Motor: Software compatibility
        46 = 1 (Name=MOTOR_WIND_CONNECT)  // Motor: Winding connection
        47 = 3 (Name=MOTOR_POLEPAIRS)  // Motor: Number of pole-pairs
      Bremsparameter:
        42 = 0 (Name=MOTOR_BRAKE_CURR_RATED, Unit=A)  // Motor holding brake: Rated current
        43 = 0 (Name=MOTOR_BRAKE_TORQ_RATED, Unit=Nm)  // Motor holding brake: Rated torque
        44 = 0 (Name=MOTOR_BRAKE_ON_TIME, Unit=s)  // Motor holding brake: Engaging delay
        45 = 0 (Name=MOTOR_BRAKE_OFF_TIME, Unit=s)  // Motor holding brake: Release delay
      Thermosensor Parameter:
        64 = 632 (Name=MOTOR_TEMPSENS_PAR1)  // Temperature sensor: Parameter 1
        65 = 2225 (Name=MOTOR_TEMPSENS_PAR2)  // Temperature sensor: Parameter 2
        66 = -30 (Name=MOTOR_TEMPSENS_PAR3)  // Temperature sensor: Parameter 3
        67 = 5.7266 (Name=MOTOR_TEMPSENS_PAR4)  // Temperature sensor: Parameter 4
        68 = 36.0938 (Name=MOTOR_TEMPSENS_PAR5)  // Temperature sensor: Parameter 5
        69 = 62.9375 (Name=MOTOR_TEMPSENS_PAR6)  // Temperature sensor: Parameter 6
        70 = 87.25 (Name=MOTOR_TEMPSENS_PAR7)  // Temperature sensor: Parameter 7
        71 = 109.6016 (Name=MOTOR_TEMPSENS_PAR8)  // Temperature sensor: Parameter 8
        72 = 130.3984 (Name=MOTOR_TEMPSENS_PAR9)  // Temperature sensor: Parameter 9
        73 = 150 (Name=MOTOR_TEMPSENS_PAR10)  // Temperature sensor: Parameter 10
      Motorparameter:
        48 = 400 (Name=MOTOR_VOLTAGE_RATED, Unit=V)  // Motor: Rated voltage
        49 = 49.22 (Name=MOTOR_VOLTAGE_CONST, Unit=mV*min)  // Motor: Voltage constant
        50 = 6000 (Name=MOTOR_SPEED_RATED, Unit=1/min)  // Motor: Rated speed
        51 = 7200 (Name=MOTOR_SPEED_MAX, Unit=1/min)  // Motor: Maximum speed
        52 = 8 (Name=MOTOR_TORQ_STALL, Unit=Nm)  // Motor: Stall torque
        53 = 6.2 (Name=MOTOR_TORQ_RATED, Unit=Nm)  // Motor: Rated torque
        54 = 33.1 (Name=MOTOR_TORQ_MAX, Unit=Nm)  // Motor: Peak torque
        55 = 0.81 (Name=MOTOR_TORQ_CONST, Unit=Nm/A)  // Motor: Torque constant
        56 = 9.83 (Name=MOTOR_CURR_STALL, Unit=A)  // Motor: Stall current
        57 = 7.62 (Name=MOTOR_CURR_RATED, Unit=A)  // Motor: Rated current
        58 = 50.83 (Name=MOTOR_CURR_MAX, Unit=A)  // Motor: Peak current
        59 = 1.31 (Name=MOTOR_WIND_CROSS_SECT, Unit=mm²)  // Motor: Line cross section
        60 = 0.9 (Name=MOTOR_STATOR_RESISTANCE, Unit=Ohm)  // Motor: Stator resistance
        61 = 0.0053 (Name=MOTOR_STATOR_INDUCTANCE, Unit=Henry)  // Motor: Stator inductance
        62 = 0.00112 (Name=MOTOR_INERTIA, Unit=kgm²)  // Motor: Moment of inertia
        63 = 0 (Name=MOTOR_COMMUT_OFFSET, Unit=rad)  // Motor: Commutation offset
        849 = 1800 (Name=MOTOR_TAU_THERM, Unit=s)  // Motor: Thermal time constant
      Isolations Parameter:
        74 = 130 (Name=MOTOR_WIND_TEMP_MAX, Unit=°C)  // Motor: Limit temperature
```

### Data object Logical/AxisObj/ggrida (Apt)

#### ggrida.apt
```
AcoposParameterTable:
  Root Parameters:
    128 = 1 (Name=SGEN_SW_END_IGNORE)  // Limit values: Ignore SW end positions
    390 = 560 (Name=UDC_NOMINAL, Unit=V)  // CTRL DC bus: Nominal voltage
    M1 (StructureEdit=FALSE)  // 8LSA55.R0045D100-1
      Allgemeine Parameter:
        30 = 16#0002 (Name=MOTOR_TYPE)  // Motor: Type
        31 = 16#0203 (Name=MOTOR_COMPATIBILITY)  // Motor: Software compatibility
        46 = 1 (Name=MOTOR_WIND_CONNECT)  // Motor: Winding connection
        47 = 4 (Name=MOTOR_POLEPAIRS)  // Motor: Number of pole-pairs
      Bremsparameter:
        42 = 0 (Name=MOTOR_BRAKE_CURR_RATED, Unit=A)  // Motor holding brake: Rated current
        43 = 0 (Name=MOTOR_BRAKE_TORQ_RATED, Unit=Nm)  // Motor holding brake: Rated torque
        44 = 0 (Name=MOTOR_BRAKE_ON_TIME, Unit=s)  // Motor holding brake: Engaging delay
        45 = 0 (Name=MOTOR_BRAKE_OFF_TIME, Unit=s)  // Motor holding brake: Release delay
      Thermosensor Parameter:
        64 = 632 (Name=MOTOR_TEMPSENS_PAR1)  // Temperature sensor: Parameter 1
        65 = 2225 (Name=MOTOR_TEMPSENS_PAR2)  // Temperature sensor: Parameter 2
        66 = -30 (Name=MOTOR_TEMPSENS_PAR3)  // Temperature sensor: Parameter 3
        67 = 5.7266 (Name=MOTOR_TEMPSENS_PAR4)  // Temperature sensor: Parameter 4
        68 = 36.0938 (Name=MOTOR_TEMPSENS_PAR5)  // Temperature sensor: Parameter 5
        69 = 62.9375 (Name=MOTOR_TEMPSENS_PAR6)  // Temperature sensor: Parameter 6
        70 = 87.25 (Name=MOTOR_TEMPSENS_PAR7)  // Temperature sensor: Parameter 7
        71 = 109.6016 (Name=MOTOR_TEMPSENS_PAR8)  // Temperature sensor: Parameter 8
        72 = 130.3984 (Name=MOTOR_TEMPSENS_PAR9)  // Temperature sensor: Parameter 9
        73 = 150 (Name=MOTOR_TEMPSENS_PAR10)  // Temperature sensor: Parameter 10
      Motorparameter:
        48 = 400 (Name=MOTOR_VOLTAGE_RATED, Unit=V)  // Motor: Rated voltage
        49 = 65.97 (Name=MOTOR_VOLTAGE_CONST, Unit=mV*min)  // Motor: Voltage constant
        50 = 4500 (Name=MOTOR_SPEED_RATED, Unit=1/min)  // Motor: Rated speed
        51 = 9000 (Name=MOTOR_SPEED_MAX, Unit=1/min)  // Motor: Maximum speed
        52 = 12.5 (Name=MOTOR_TORQ_STALL, Unit=Nm)  // Motor: Stall torque
        53 = 9.5 (Name=MOTOR_TORQ_RATED, Unit=Nm)  // Motor: Rated torque
        54 = 41.4 (Name=MOTOR_TORQ_MAX, Unit=Nm)  // Motor: Peak torque
        55 = 1.09 (Name=MOTOR_TORQ_CONST, Unit=Nm/A)  // Motor: Torque constant
        56 = 11.46 (Name=MOTOR_CURR_STALL, Unit=A)  // Motor: Stall current
        57 = 8.71 (Name=MOTOR_CURR_RATED, Unit=A)  // Motor: Rated current
        58 = 47.29 (Name=MOTOR_CURR_MAX, Unit=A)  // Motor: Peak current
        59 = 1.97 (Name=MOTOR_WIND_CROSS_SECT, Unit=mm²)  // Motor: Line cross section
        60 = 0.51 (Name=MOTOR_STATOR_RESISTANCE, Unit=Ohm)  // Motor: Stator resistance
        61 = 0.00496 (Name=MOTOR_STATOR_INDUCTANCE, Unit=Henry)  // Motor: Stator inductance
        62 = 0.000819 (Name=MOTOR_INERTIA, Unit=kgm²)  // Motor: Moment of inertia
        63 = 0 (Name=MOTOR_COMMUT_OFFSET, Unit=rad)  // Motor: Commutation offset
        849 = 2400 (Name=MOTOR_TAU_THERM, Unit=s)  // Motor: Thermal time constant
      Isolations Parameter:
        74 = 130 (Name=MOTOR_WIND_TEMP_MAX, Unit=°C)  // Motor: Limit temperature
```

### Data object Logical/AxisObj/gbuffera (Apt)

#### gbuffera.apt
```
AcoposParameterTable:
  Root Parameters:
    128 = 1 (Name=SGEN_SW_END_IGNORE, Disabled=TRUE)  // Limit values: Ignore SW end positions
    390 = 560 (Name=UDC_NOMINAL, Unit=V)  // CTRL DC bus: Nominal voltage
    M1 (StructureEdit=FALSE)  // 8LSA55.R0045D200-1
      Allgemeine Parameter:
        30 = 16#0002 (Name=MOTOR_TYPE)  // Motor: Type
        31 = 16#0203 (Name=MOTOR_COMPATIBILITY)  // Motor: Software compatibility
        46 = 1 (Name=MOTOR_WIND_CONNECT)  // Motor: Winding connection
        47 = 4 (Name=MOTOR_POLEPAIRS)  // Motor: Number of pole-pairs
      Bremsparameter:
        42 = 1 (Name=MOTOR_BRAKE_CURR_RATED, Unit=A)  // Motor holding brake: Rated current
        43 = 15 (Name=MOTOR_BRAKE_TORQ_RATED, Unit=Nm)  // Motor holding brake: Rated torque
        44 = 0.05 (Name=MOTOR_BRAKE_ON_TIME, Unit=s)  // Motor holding brake: Engaging delay
        45 = 0.05 (Name=MOTOR_BRAKE_OFF_TIME, Unit=s)  // Motor holding brake: Release delay
      Thermosensor Parameter:
        64 = 632 (Name=MOTOR_TEMPSENS_PAR1)  // Temperature sensor: Parameter 1
        65 = 2225 (Name=MOTOR_TEMPSENS_PAR2)  // Temperature sensor: Parameter 2
        66 = -30 (Name=MOTOR_TEMPSENS_PAR3)  // Temperature sensor: Parameter 3
        67 = 5.7266 (Name=MOTOR_TEMPSENS_PAR4)  // Temperature sensor: Parameter 4
        68 = 36.0938 (Name=MOTOR_TEMPSENS_PAR5)  // Temperature sensor: Parameter 5
        69 = 62.9375 (Name=MOTOR_TEMPSENS_PAR6)  // Temperature sensor: Parameter 6
        70 = 87.25 (Name=MOTOR_TEMPSENS_PAR7)  // Temperature sensor: Parameter 7
        71 = 109.6016 (Name=MOTOR_TEMPSENS_PAR8)  // Temperature sensor: Parameter 8
        72 = 130.3984 (Name=MOTOR_TEMPSENS_PAR9)  // Temperature sensor: Parameter 9
        73 = 150 (Name=MOTOR_TEMPSENS_PAR10)  // Temperature sensor: Parameter 10
      Motorparameter:
        48 = 400 (Name=MOTOR_VOLTAGE_RATED, Unit=V)  // Motor: Rated voltage
        49 = 65.97 (Name=MOTOR_VOLTAGE_CONST, Unit=mV*min)  // Motor: Voltage constant
        50 = 4500 (Name=MOTOR_SPEED_RATED, Unit=1/min)  // Motor: Rated speed
        51 = 9000 (Name=MOTOR_SPEED_MAX, Unit=1/min)  // Motor: Maximum speed
        52 = 12.5 (Name=MOTOR_TORQ_STALL, Unit=Nm)  // Motor: Stall torque
        53 = 9.5 (Name=MOTOR_TORQ_RATED, Unit=Nm)  // Motor: Rated torque
        54 = 41.4 (Name=MOTOR_TORQ_MAX, Unit=Nm)  // Motor: Peak torque
        55 = 1.09 (Name=MOTOR_TORQ_CONST, Unit=Nm/A)  // Motor: Torque constant
        56 = 11.46 (Name=MOTOR_CURR_STALL, Unit=A)  // Motor: Stall current
        57 = 8.71 (Name=MOTOR_CURR_RATED, Unit=A)  // Motor: Rated current
        58 = 47.29 (Name=MOTOR_CURR_MAX, Unit=A)  // Motor: Peak current
        59 = 1.97 (Name=MOTOR_WIND_CROSS_SECT, Unit=mm²)  // Motor: Line cross section
        60 = 0.51 (Name=MOTOR_STATOR_RESISTANCE, Unit=Ohm)  // Motor: Stator resistance
        61 = 0.00496 (Name=MOTOR_STATOR_INDUCTANCE, Unit=Henry)  // Motor: Stator inductance
        62 = 0.000819 (Name=MOTOR_INERTIA, Unit=kgm²)  // Motor: Moment of inertia
        63 = 0 (Name=MOTOR_COMMUT_OFFSET, Unit=rad)  // Motor: Commutation offset
        849 = 2400 (Name=MOTOR_TAU_THERM, Unit=s)  // Motor: Thermal time constant
      Isolations Parameter:
        74 = 130 (Name=MOTOR_WIND_TEMP_MAX, Unit=°C)  // Motor: Limit temperature
```

### Data object Logical/AxisObj/gcatchba (Apt)

#### gcatchba.apt
```
AcoposParameterTable:
  Root Parameters:
    128 = 1 (Name=SGEN_SW_END_IGNORE)  // Limit values: Ignore SW end positions
    390 = 560 (Name=UDC_NOMINAL, Unit=V)  // CTRL DC bus: Nominal voltage
    M1 (StructureEdit=FALSE)  // 8LSA35.R2030D000-3
      Allgemeine Parameter:
        30 = 16#0002 (Name=MOTOR_TYPE)  // Motor: Type
        31 = 16#0203 (Name=MOTOR_COMPATIBILITY)  // Motor: Software compatibility
        46 = 1 (Name=MOTOR_WIND_CONNECT)  // Motor: Winding connection
      Bremsparameter:
        42 = 0 (Name=MOTOR_BRAKE_CURR_RATED, Unit=A)  // Motor holding brake: Rated current
        43 = 0 (Name=MOTOR_BRAKE_TORQ_RATED, Unit=Nm)  // Motor holding brake: Rated torque
        44 = 0 (Name=MOTOR_BRAKE_ON_TIME, Unit=s)  // Motor holding brake: Engaging delay
        45 = 0 (Name=MOTOR_BRAKE_OFF_TIME, Unit=s)  // Motor holding brake: Release delay
      Thermosensor Parameter:
        64 = 632 (Name=MOTOR_TEMPSENS_PAR1)  // Temperature sensor: Parameter 1
        65 = 2225 (Name=MOTOR_TEMPSENS_PAR2)  // Temperature sensor: Parameter 2
        66 = -30 (Name=MOTOR_TEMPSENS_PAR3)  // Temperature sensor: Parameter 3
        67 = 5.7266 (Name=MOTOR_TEMPSENS_PAR4)  // Temperature sensor: Parameter 4
        68 = 36.0938 (Name=MOTOR_TEMPSENS_PAR5)  // Temperature sensor: Parameter 5
        69 = 62.9375 (Name=MOTOR_TEMPSENS_PAR6)  // Temperature sensor: Parameter 6
        70 = 87.25 (Name=MOTOR_TEMPSENS_PAR7)  // Temperature sensor: Parameter 7
        71 = 109.6016 (Name=MOTOR_TEMPSENS_PAR8)  // Temperature sensor: Parameter 8
        72 = 130.3984 (Name=MOTOR_TEMPSENS_PAR9)  // Temperature sensor: Parameter 9
        73 = 150 (Name=MOTOR_TEMPSENS_PAR10)  // Temperature sensor: Parameter 10
      Motorparameter:
        47 = 4 (Name=MOTOR_POLEPAIRS)  // Motor: Number of pole-pairs
        48 = 400 (Name=MOTOR_VOLTAGE_RATED, Unit=V)  // Motor: Rated voltage
        49 = 87.96 (Name=MOTOR_VOLTAGE_CONST, Unit=mV*min)  // Motor: Voltage constant
        50 = 3000 (Name=MOTOR_SPEED_RATED, Unit=1/min)  // Motor: Rated speed
        51 = 9000 (Name=MOTOR_SPEED_MAX, Unit=1/min)  // Motor: Maximum speed
        52 = 2.3 (Name=MOTOR_TORQ_STALL, Unit=Nm)  // Motor: Stall torque
        53 = 2.1 (Name=MOTOR_TORQ_RATED, Unit=Nm)  // Motor: Rated torque
        54 = 9.2 (Name=MOTOR_TORQ_MAX, Unit=Nm)  // Motor: Peak torque
        55 = 1.45 (Name=MOTOR_TORQ_CONST, Unit=Nm/A)  // Motor: Torque constant
        56 = 1.6 (Name=MOTOR_CURR_STALL, Unit=A)  // Motor: Stall current
        57 = 1.4 (Name=MOTOR_CURR_RATED, Unit=A)  // Motor: Rated current
        58 = 6.8 (Name=MOTOR_CURR_MAX, Unit=A)  // Motor: Peak current
        59 = 0.181 (Name=MOTOR_WIND_CROSS_SECT, Unit=mm²)  // Motor: Line cross section
        60 = 12.2 (Name=MOTOR_STATOR_RESISTANCE, Unit=Ohm)  // Motor: Stator resistance
        61 = 0.063 (Name=MOTOR_STATOR_INDUCTANCE, Unit=Henry)  // Motor: Stator inductance
        62 = 9E-05 (Name=MOTOR_INERTIA, Unit=kgm²)  // Motor: Moment of inertia
        63 = 0 (Name=MOTOR_COMMUT_OFFSET, Unit=rad)  // Motor: Commutation offset
      Isolations Parameter:
        74 = 130 (Name=MOTOR_WIND_TEMP_MAX, Unit=°C)  // Motor: Limit temperature
      849 = 2040 (Name=MOTOR_TAU_THERM, Unit=s)  // Motor: Thermal time constant
```

### Data object Logical/AxisObj/gunwfeeda (Apt)

#### gunwfeeda.apt
```
AcoposParameterTable:
  Root Parameters:
    45 = 1 (Name=MOTOR_BRAKE_OFF_TIME, Unit=s)  // Motor holding brake: Release delay
    230 = PCTRL_S_SET (Name=PCTRL_S_ACT_PARID)  // CTRL Position controller: Actual encoder position parameter ID
    64201 = 126562 (Name=SERVO_V_MAX_OUTPUT, Unit=Units/s)  // Servo drive adjustment: Velocity at maximum output value
    128 = 1 (Name=SGEN_SW_END_IGNORE)  // Limit values: Ignore SW end positions
    90 = 77 (Name=BRAKE_MODE)  // Motor holding brake: Mode
    44 = 1 (Name=MOTOR_BRAKE_ON_TIME, Unit=s)  // Motor holding brake: Engaging delay
```

### Data object Logical/AxisObj/gsafetya (Apt)

#### gsafetya.apt
```
AcoposParameterTable:
  Root Parameters:
    128 = 1 (Name=SGEN_SW_END_IGNORE)  // Limit values: Ignore SW end positions
    390 = 560 (Name=UDC_NOMINAL, Unit=V)  // CTRL DC bus: Nominal voltage
```

### Data object Logical/AxisObj/gPackBelta (Apt)

#### gPackBelta.apt
```
AcoposParameterTable:
  Root Parameters:
    230 = PCTRL_S_SET (Name=PCTRL_S_ACT_PARID)
    64201 = 546116,666666667 (Name=SERVO_V_MAX_OUTPUT, Unit=Units/s)  // Servo drive adjustment: Velocity at maximum output value
    128 = 3 (Name=SGEN_SW_END_IGNORE)  // Limit values: Ignore SW end positions
```

### RCP_Tool.typ - Package data types
```iecst
(********************************************************************
 * COPYRIGHT -- Bernecker + Rainer
 ********************************************************************
 * File: RCP_Tool.typ
 * Author: beutert
 * Created: September 03, 2012
 ********************************************************************
 * Global data types of project csv_bsp
 ********************************************************************)

TYPE
	rcp_tool_typ : 	STRUCT
		description : STRING[80]; (*Beschreibung*)
		addSupportSpindle : BOOL; (*Zusätzliche Stützwelle*)
		cogCutting : UINT; (*Zahnrad Stanzwerkzeug*)
		cogSupportSpindle : UINT; (*Zahnrad Stützwelle*)
		numberToolSegments : USINT; (*Anzahl der Nutzen / Werkzeugumfang*)
		cutStartPosition : DINT; (*Anfangsposition Schnitt innerhalb einer Nutzenperiode [um]*)
		cutEndPosition : DINT; (*Endposition Schnitt innerhalb einer Nutzenperiode [um]*)
		homePosition : REAL; (*Referenzposition der Achse [um]*)
		cogmodul:REAL := 3175.0; (* in mikrometer *)
		gearRatioMotor :UINT := 5;
	END_STRUCT;
	TOOL_Hndl_typ : 	STRUCT
		ReqParaRead : BOOL;
		ReqParaWrite : BOOL;
		ReqParaWriteAfterValueChanged : BOOL;
		ReqDirRead : BOOL;
		ReqCreateNew : BOOL;
		ReqNewRecipe : BOOL;
		ReqDelRecipe : BOOL;
		ReqSaveAs : BOOL;
		ReqSaveRecipeAs : BOOL;
		BtnNew : BOOL;
		BtnSaveAs : BOOL;
		SetListBoxIdxToZero : BOOL;
		ListboxMaxLines : UINT;
		ListboxFileNames : ARRAY[0..99]OF STRING[46];
		ListboxIdx : UINT;
		LayerMessageBoxOverwrite : USINT; (*switches the layer on or off*)
		LayerMessageBoxDeleteFile : USINT; (*switches the layer on or off*)
		LayerNewFileName : USINT; (*switches the layer on or off*)
		LayerMessageBoxSaveFile : USINT; (*switches the layer on or off*)
		StatusNewFileName : UINT;
		NewFileNameEntered : BOOL; (*completion datapoint for filename*)
		FileOverWrite : USINT; (*answer from messagebox*)
		FileDelete : USINT; (*answer from messagebox*)
		FileNameNew : STRING[80];
		FileNameSave : STRING[80];
		FileNameDelete : STRING[80];
		FileNameSelected : STRING[80];
		ListBoxMaxIdx : UINT;
		OverwriteFile : BOOL; (*when save was selected, don't ask for overwrite, do it*)
		ValueChanged : BOOL; (*true if any value displayed on the page was changed*)
		ScrollUpLbo1 : USINT;
		ScrollDownLbo1 : USINT;
		ScrollHomeLbo1 : USINT;
		ScrollEndLbo1 : USINT;
		ScrollUpLbo2 : USINT;
		ScrollDownLbo2 : USINT;
		ScrollHomeLbo2 : USINT;
		ScrollEndLbo2 : USINT;
		StatusBmp : UINT;
		DeleteFileYes : USINT;
		DeleteFileNo : USINT;
		SaveFileYes : USINT;
		SaveFileNo : USINT;
		OverwriteFileYes : USINT;
		OverwriteFileNo : USINT;
	END_STRUCT;
END_TYPE
```

### RCP_Prog.typ - Package data types
```iecst
(********************************************************************
 * COPYRIGHT -- Bernecker + Rainer
 ********************************************************************
 * File: RCP_Prog.typ
 * Author: beutert
 * Created: September 03, 2012
 ********************************************************************
 * Global data types of project csv_bsp
 ********************************************************************)
(*======================================================================================================================================*)
(*APPLICATION RECIPE DATA*)
(*======================================================================================================================================*)

TYPE
	rcp_prog_typ : 	STRUCT  (*Program/recipe parameters*)
		header : rcp_prog_header_typ; (*File header for recipe information*)
		general : rcp_prog_general_typ;
		dancer : rcp_prog_dancer_typ;
		tensionMeas : rcp_prog_tensMeas_typ;
		cutUnit1 : rcp_prog_cutUnit_typ;
		cutUnit2 : rcp_prog_cutUnit_typ;
		cutUnit3 : rcp_prog_cutUnit_typ;
		UnwinderOpSide : rcp_prog_wind_typ;
		UnwinderDrvSide : rcp_prog_wind_typ;
		mainUnwind : rcp_prog_wind_typ;
		grid1 : rcp_prog_wind_typ;
		grid2 : rcp_prog_wind_typ;
		gridwinderleft : rcp_prog_wind_typ;
		gridwinderright : rcp_prog_wind_typ;
		laminator1 : rcp_prog_wind_typ;
		laminator2 : rcp_prog_wind_typ;
		LaminatorRegist : rcp_prog_laminatorReg_typ; (* Struktur für den Laminator bzw. Laminierer*)
		spender1 : rcp_prog_spend_typ;
		spender2 : rcp_prog_spend_typ;
		spender3 : rcp_prog_spend_typ; (*winder: FB_WinderData;*)
		longCut : rcp_prog_conveyor_data_typ;
		conveyor : rcp_prog_conveyor_data_typ;
		longcutter : rcp_prog_conveyor_data_typ;
		pullbelt : rcp_prog_conveyor_data_typ;
		catchbelt : rcp_prog_conveyor_data_typ;
		endModule : rcp_prog_endModule_typ;
	END_STRUCT;
	rcp_prog_header_typ : 	STRUCT  (*Header for program/recipe information*)
		name : ARRAY[0..RCP_PROG_TEXT_FILENAME_MAX]OF UINT; (*Name des Program/Rezept*)
		description : ARRAY[0..RCP_PROG_TEXT_DESCRIPTION_MAX]OF UINT; (*Zusätzliche Beschreibung*)
		changed : USINT; (*Rezept wurde geändert*)
	END_STRUCT;
	rcp_prog_general_typ : 	STRUCT  (*general data*)
		masterDeceleration : REAL; (*deceleration [units/s² = µm/s²] of virtual amster axis*)
		masterAcceleration : REAL; (*acceleration [units/s² = µm/s²] of virtual amster axis*)
		periodLength : REAL; (*Material period [µm]*)
		startVelocity : REAL; (*start velocity [units/s]*)
		maxVelocity : REAL; (*maximum product velocity [units/s]*)
		lenght1 : REAL;
		speedToCycleWebturrit : REAL;
		lenght2 : REAL;
	END_STRUCT;
	rcp_prog_dancer_typ : 	STRUCT  (*dancer settings*)
		radiusCtrlOn : BOOL; (*Radius control On/Off*)
		cylinderTension : BOOL; (*Tension On/Off*)
		force : REAL; (*dancer force via prop ventile [%]*)
	END_STRUCT;
	rcp_prog_wind_typ : 	STRUCT  (*main unwinding unit settings*)
		warnDiam : UDINT;
		stopDiam : UDINT;
		minDiamTension : UDINT;
		maxDiamTension : UDINT;
		mode : UDINT;
		reverse : BOOL;
	END_STRUCT;
	rcp_prog_tensMeas_typ : 	STRUCT  (*web tension measurement unit settings*)
		mode : UDINT; (*Mode*)
		webTension : REAL; (*Web tension *)
	END_STRUCT;
	rcp_prog_cutUnit_typ : 	STRUCT  (*cut unit settings*)
		mode : UDINT; (*Mode*)
		toolfilename : STRING[80]; (*name of tool file*)
		toolNumber : USINT; (*Tool number*)
		markPointNo : USINT; (*number of mark point (index?)*)
		tool : rcp_tool_typ; (*selected tool parameter*)
		RmWindow : REAL; (*Range before / after the expected position in which the trigger signal may occur [Master Units]*)
		RmOffset : REAL; (*Reg mark position relative to cut position [Master Units]*)
		Insetting : REAL; (*Insetting ratio [%] (100% means the velocity in the cam equals the velocity in the compensation gear)*)
		MaxCorr : REAL; (*Insetting ratio [%] (100% means the velocity in the cam equals the velocity in the compensation gear)*)
	END_STRUCT;
	rcp_prog_laminatorReg_typ : 	STRUCT
		mode : UDINT; (*Mode*)
		Winder : rcp_prog_wind_typ; (*torque setpoint at minimum diameter [Nm]*)
		Unwinder : rcp_prog_wind_typ; (*torque setpoint at maximum diameter [Nm]*)
		reverse : BOOL; (*TRUE = reverse direction*)
		LabelPeriod : REAL; (*Label dispenser period/ Rapportlänge der Spendeetiketten*)
		ProductLenghtMaster : REAL; (*Product lenght on master axis/ Periodenlänge der Spendeetiketten auf der Hauptbahn*)
		RegMarkPos : REAL; (*Abstand zwischen Registermarke und Spendeposition*)
		LabelOffset : REAL; (*Label offset relative to start position/ Offset der Länge zwischen Labelbahnsensor und Spendeposition*)
	END_STRUCT;
	rcp_prog_spend_typ : 	STRUCT  (*spender (unwinder/winder) settings*)
		mode : UDINT; (*Mode*)
		minDiamTorq : REAL; (*torque setpoint at minimum diameter [Nm]*)
		maxDiamTorq : REAL; (*torque setpoint at maximum diameter [Nm]*)
		reverse : BOOL; (*TRUE = reverse direction*)
		LabelPeriod : REAL; (*Label dispenser period/ Rapportlänge der Spendeetiketten*)
		ProductLenghtMaster : REAL; (*Product lenght on master axis/ Periodenlänge der Spendeetiketten auf der Hauptbahn*)
		RegMarkPos : REAL; (*Abstand zwischen Registermarke und Spendeposition*)
		LabelOffset : REAL; (*Label offset relative to start position/ Offset der Länge zwischen Labelbahnsensor und Spendeposition*)
	END_STRUCT;
	rcp_prog_lamin_typ : 	STRUCT  (*spender (unwinder/winder) settings*)
		mode : UDINT; (*Mode*)
		minDiamTorq : REAL; (*torque setpoint at minimum diameter [Nm]*)
		maxDiamTorq : REAL; (*torque setpoint at maximum diameter [Nm]*)
		reverse : BOOL; (*TRUE = reverse direction*)
		LabelPeriod : REAL; (*Label dispenser period/ Rapportlänge der Spendeetiketten*)
		ProductLenghtMaster : REAL; (*Product lenght on master axis/ Periodenlänge der Spendeetiketten auf der Hauptbahn*)
		RegMarkPos : REAL; (*Abstand zwischen Registermarke und Spendeposition*)
		LabelOffset : REAL; (*Label offset relative to start position/ Offset der Länge zwischen Labelbahnsensor und Spendeposition*)
	END_STRUCT;
	rcp_prog_longCut_typ : 	STRUCT  (*long cut unit settings*)
		mode : UDINT; (*Mode*)
		veloRelative : REAL; (*relative velocity to master [%]*)
	END_STRUCT;
	rcp_prog_conveyor_data_typ : 	STRUCT
		setvaluevisu : REAL;
		offsetOnOff : BOOL;
		mode : UDINT;
		setPieces : UINT;
		validPieces : UINT;
		sensor1 : INT;
		sensor2 : INT;
		sensor3 : INT;
		sensor4 : INT;
		sensor5 : INT;
		sensor6 : INT;
		sensor7 : INT;
		sensor8 : INT;
		sensor9 : INT;
	END_STRUCT;
	rcp_prog_endModule_typ : 	STRUCT  (*settings for end module (belts and tandem winder)*)
		mode : UDINT; (*Mode*)
		minDiamPressureTop : REAL; (*pressure at minimum diameter top winder [%]*)
		maxDiamPressureTop : REAL; (*pressure at maximum diameter top winder [%]*)
		minDiamPressureBot : REAL; (*pressure at minimum diameter bottom winder [%]*)
		maxDiamPressureBot : REAL; (*pressure at maximum diameter bottom winder [%]*)
		minDiamTensionTop : REAL; (*tension force at minimum diameter top winder [N]*)
		maxDiamTensionTop : REAL; (*tension force at maximum diameter top winder [N]*)
		minDiamValueTop : REAL; (*corresponding minimum diameter value top winder [µm]*)
		reverseTopWind : BOOL; (*TRUE = reverse direction of top winder*)
		minDiamTensionBot : REAL; (*tension force at minimum diameter bottom winder [N]*)
		maxDiamTensionBot : REAL; (*tension force at maximum diameter bottom winder [N]*)
		minDiamValueBot : REAL; (*corresponding minimum diameter value bottom winder [µm]*)
		reverseBotWind : BOOL; (*TRUE = reverse direction of bottom winder*)
		veloRelativeTopBelt : REAL; (*relative velocity to master [%]*)
		veloRelativeConvBelt : REAL; (*relative velocity to master [%]*)
		veloBatchConvBelt : REAL; (*Batch velocity to master [%]*)
		batchDistance : REAL; (*relative velocity to master [%]*)
		numberPapers : UDINT; (*number of Papers in batch*)
	END_STRUCT;
END_TYPE

(*======================================================================================================================================*)
(*CSV FILE HANDLING DATA TYPES*)
(*======================================================================================================================================*)

TYPE
	CSVHndl_typ : 	STRUCT
		ReqParaRead : BOOL;
		ReqParaWrite : BOOL;
		ReqParaWriteAfterValueChanged : BOOL;
		ReqDirRead : BOOL;
		ReqCreateNew : BOOL;
		ReqNewRecipe : BOOL;
		ReqDelRecipe : BOOL;
		ReqSaveAs : BOOL;
		ReqSaveRecipeAs : BOOL;
		BtnNew : BOOL;
		BtnSaveAs : BOOL;
		SetListBoxIdxToZero : BOOL;
		ListBoxRecipeChanged : BOOL; (*when another recipe was selected*)
		ListboxMaxLines : UINT;
		ListboxFileNames : ARRAY[0..99]OF STRING[46];
		ListboxIdx : UINT;
		LayerMessageBoxOverwrite : USINT; (*switches the layer on or off*)
		LayerMessageBoxDeleteFile : USINT; (*switches the layer on or off*)
		LayerNewFileName : USINT; (*switches the layer on or off*)
		LayerMessageBoxSaveFile : USINT; (*switches the layer on or off*)
		LayersProgPara : ARRAY[0..20]OF USINT; (*switches the layer on or off*)
		ListboxProgParaIdx : UINT;
		ListboxProgParaMaxLines : UINT := 15;
		StatusNewFileName : UINT;
		NewFileNameEntered : BOOL; (*completion datapoint for filename*)
		FileOverWrite : USINT; (*answer from messagebox*)
		FileDelete : USINT; (*answer from messagebox*)
		FileNameNew : STRING[80];
		FileNameSave : STRING[80];
		FileNameDelete : STRING[80];
		FileNameSelected : STRING[80];
		ListBoxMaxIdx : UINT;
		OverwriteFile : BOOL; (*when save was selected, don't ask for overwrite, do it*)
		ValueChanged : BOOL; (*true if any value displayed on the page was changed*)
		ToolSelectedCutU1 : BOOL; (*a tool file was selected from the list*)
		ToolSelectedCutU2 : BOOL; (*a tool file was selected from the list*)
		ToolSelectedCutU3 : BOOL; (*a tool file was selected from the list*)
		ScrollUpLbo1 : USINT;
		ScrollDownLbo1 : USINT;
		ScrollHomeLbo1 : USINT;
		ScrollEndLbo1 : USINT;
		ScrollUpLbo2 : USINT;
		ScrollDownLbo2 : USINT;
		ScrollHomeLbo2 : USINT;
		ScrollEndLbo2 : USINT;
		ScrollUpLbo3 : USINT;
		ScrollDownLbo3 : USINT;
		ScrollHomeLbo3 : USINT;
		ScrollEndLbo3 : USINT;
		DeleteFileYes : USINT;
		DeleteFileNo : USINT;
		SaveFileYes : USINT;
		SaveFileNo : USINT;
		OverwriteFileYes : USINT;
		OverwriteFileNo : USINT;
		StatusBmpRadiusCtrlOnOff : UINT;
		StatusBmpTensionOnOff : UINT;
		StatusBmpReverseGeneral : UINT;
		StatusBmpReverseUnwinder : UINT;
		StatusBmpReverseTensMeas : UINT;
		StatusBmpReverseLongCut : UINT;
		StatusBmpReverseSpender1 : UINT;
		StatusBmpReverseGrid1 : UINT;
		StatusBmpReverseSpender2 : UINT;
		StatusBmpReverseGrid2 : UINT;
		StatusBmpReverseWindTop : UINT;
		StatusBmpReverseWindBot : UINT;
		StatusBmpReverseConvey : UINT;
		StatusBmpFoundFileCutU1 : UINT;
		StatusBtnRefreshCutU1 : UINT;
		StatusBmpFoundFileCutU2 : UINT;
		StatusBtnRefreshCutU2 : UINT;
		StatusBmpFoundFileCutU3 : UINT;
		StatusBtnRefreshCutU3 : UINT;
	END_STRUCT;
END_TYPE
```

### RCP_Glob.typ - Package data types
```iecst
(********************************************************************
 * COPYRIGHT -- Bernecker + Rainer
 ********************************************************************
 * File: RCP_Glob.typ
 * Author: beutert
 * Created: September 07, 2012
 *
 * History:
 * 2012-09-20 /schoenefeldr/
 * 		Added linearisation parameters for diameter sensors to recipe
 *
 *
 *
 ********************************************************************
 * Global data types of project csv_bsp
 ********************************************************************)
(*======================================================================================================================================*)
(*GENERAL DATA*)
(*======================================================================================================================================*)

TYPE
	Button_typ : 	STRUCT
		F1 : USINT;
		F2 : USINT;
		F3 : USINT;
		F4 : USINT;
		F5 : USINT;
		F6 : USINT;
		F7 : USINT;
		F8 : USINT;
		F9 : USINT;
		F10 : USINT;
		F11 : USINT;
		F12 : USINT;
		Status : ARRAY[0..12]OF UINT;
	END_STRUCT;
END_TYPE

(*======================================================================================================================================*)
(*MACHINE RECIPE DATA*)
(*======================================================================================================================================*)

TYPE
	rcp_machine_Wind_Type : 	STRUCT  (*Diameter offsets and additional sensor parameters*)
		DiamOffsMainUnw : REAL; (*Diameter offset value (distance from sensor to core) [mm]*)
		DiamOffsGrid1 : REAL; (*Diameter offset value (distance from sensor to core) [mm]*)
		DiamOffsGrid2 : REAL; (*Diameter offset value (distance from sensor to core) [mm]*)
		DiamOffsLaminator1 : REAL;
		DiamOffsLaminator2 : REAL;
		DiamOffsSpend1 : REAL; (*Diameter offset value (distance from sensor to core) [mm]*)
		DiamOffsSpend2 : REAL; (*Diameter offset value (distance from sensor to core) [mm]*)
		DiamOffsSpend3 : REAL; (*Diameter offset value (distance from sensor to core) [mm]*)
		DiamOffsSpend4 : REAL; (*Diameter offset value (distance from sensor to core) [mm]*)
		DiamOffsTopTWind : REAL; (*Diameter offset value (distance from sensor to core) [mm]*)
		DiamOffsBotTWind : REAL; (*Diameter offset value (distance from sensor to core) [mm]*)
		CoreDiam : REAL; (*Diameter of core [mm]*)
		CoreMaxDiamSensor : REAL; (*Maximum value for diameter sensor value [mm]*)
		CoreMinDiamSensor : REAL; (*Minimum value for diameter sensor value [mm]*)
		UseDiamLinearCorr : BOOL; (*Apply linear correction for diameter sensors*)
		DiamCorrGain : REAL; (*Gain for linear diameter correction [1]*)
		DiamCorrOffs : REAL; (*Offset for linear diameter correction [mm]*)
	END_STRUCT;
	rcp_machine_general_typ : 	STRUCT  (*General machine data*)
		max_diameter : REAL; (*maximum coil diameter*)
		model_type : INT; (*Machine model type 1=herpa_print*)
		MatPeriodMin : REAL;
		MatPeriodMax : REAL;
		spraygap	: REAL;
		spraytime	:REAL;
	END_STRUCT;
	rcp_machine_unwind_typ : 	STRUCT  (*Diameter values for winders*)
		coreDiam : USINT;
		frictionCompensation : USINT;
		velocityOverride : USINT;
		GEAR_RATIO : USINT;
		StopDiam : UDINT; (*Diameter value for stop [mm]*)
		WarnDiam : REAL; (*Diameter value for warning [mm]*)
		DistanceToRmSensor : REAL; (*Diameter value for warning [mm]*)
		DistanceToLabelSensor : REAL; (*Diameter value for warning [mm]*)
	END_STRUCT;
	rcp_machine_LaminatorReg_typ : 	STRUCT  (*Diameter values for winders*)
		WinderStopDiam : REAL; (*Diameter value for stop [mm]*)
		WinderWarnDiam : REAL; (*Diameter value for warning [mm]*)
		UnwinderStopDiam : REAL; (*Diameter value for stop [mm]*)
		UnwinderWarnDiam : REAL; (*Diameter value for warning [mm]*)
		DistanceToRmSensor : REAL; (*Diameter value for warning [mm]*)
		DistanceToLaminatprSensor : REAL; (*Diameter value for warning [mm]*)
	END_STRUCT;
	rcp_machine_twind_typ : 	STRUCT  (*machine recipe parameters for tandem winder*)
		StopDiam : REAL; (*Diameter value for stop [mm]*)
		WarnDiam : REAL; (*Diameter value for warning [mm]*)
		frictionCompensation : REAL; (*friction compensation [Nm] (on motor side)*)
		MinPressure : REAL; (*Valve pressure at minimum diameter [%]*)
		MaxPressure : REAL; (*Valve pressure at stop diameter [%]*)
		VelocityOverride : REAL; (*Velocity override [%]*)
	END_STRUCT;
	rcp_machine_markp_typ : 	STRUCT  (*machine parameters for markpoints (registration marks)*)
		position : DINT; (*markpoint sensor position [mm]*)
	END_STRUCT;
	rcp_machine_cutUnit_typ : 	STRUCT  (*machine parameters for cutting units*)
		position : DINT; (*cutting unit position [mm]*)
	END_STRUCT;
	rcp_machine_pullBrakeUnit_typ : 	STRUCT  (*machine parameters for pull brake unit*)
		gearOverride : REAL; (*gear ratio override [%]*)
	END_STRUCT;
	rcp_machine_typ : 	STRUCT  (*Machine description*)
		general : rcp_machine_general_typ; (*structure for general data and settings*)
		Winders : rcp_machine_Wind_Type; (*offset settings for diameter sensors*)
		UnwinderOpSide : rcp_machine_unwind_typ; (*settings for main unwinder*)
		mainUnwind : rcp_machine_unwind_typ; (*settings for main unwinder*)
		UnwinderDrvSide : rcp_machine_unwind_typ; (*settings for main unwinder*)
		laminatorReg : rcp_machine_LaminatorReg_typ;
		pbu : rcp_machine_pullBrakeUnit_typ; (*settings for pull brake unit*)
		cut1 : rcp_machine_cutUnit_typ; (*settings for cut unit 1*)
		cut2 : rcp_machine_cutUnit_typ; (*settings for cut unit 2*)
		cut3 : rcp_machine_cutUnit_typ; (*settings for cut unit 2*)
		markpoint1 : rcp_machine_markp_typ; (*settings for markpoint sensor 1*)
		markpoint2 : rcp_machine_markp_typ; (*settings for markpoint sensor 2*)
		markpoint3 : rcp_machine_markp_typ; (*settings for markpoint sensor 2*)
		grid1 : rcp_machine_unwind_typ; (*settings for grid winder 1*)
		grid2 : rcp_machine_unwind_typ; (*settings for grid winder 2*)
		gridwinderleft : rcp_machine_unwind_typ; (*settings for grid winder 2*)
		gridwinderright : rcp_machine_unwind_typ; (*settings for grid winder 2*)
		laminator1 : rcp_machine_unwind_typ; (*settings for grid winder 2*)
		laminator2 : rcp_machine_unwind_typ; (*settings for grid winder 2*)
		spender1 : rcp_machine_unwind_typ; (*settings for spender 1*)
		spender2 : rcp_machine_unwind_typ; (*settings for spender 2*)
		spender3 : rcp_machine_unwind_typ; (*settings for spender 3 (additional winder)*)
		topTandemWind : rcp_machine_twind_typ; (*settings for top tandem winder*)
		botTandemWind : rcp_machine_twind_typ; (*settings for bottom tandem winder*)
	END_STRUCT;
	rcp_cutting_typ : 	STRUCT
		machdata : rcp_machine_cutUnit_typ;
		recipe : rcp_prog_cutUnit_typ;
	END_STRUCT;
END_TYPE

(*======================================================================================================================================*)
(*GENERAL RECIPE DATA STRUCTURES*)
(*======================================================================================================================================*)

TYPE
	CSV_Header_typ : 	STRUCT
		CustomerName : STRING[80];
		MachineNumber : STRING[80];
		SW_Version : STRING[80];
	END_STRUCT;
END_TYPE
```
